(* Logix 5000 project; controller reports 1756-L63 rev 20.11; software revision 20.04; part 11 of 52 *)

        [254].log_data[16].valid := 1, [254].log_data[17].valid := 1, [254].log_data[18].valid := 1, [254].log_data[19].valid := 1, [254].time.Year := 2023, [254].time.Month := 1, [254].time.Day := 18, [254].time.Hour := 21, [254].time.Minute := 34, [254].time.Second := 59, [255].log_data[0].min := 1.0, [255].log_data[0].max := 1.0, [255].log_data[0].total := 300.0, [255].log_data[0].time := 300.0, [255].log_data[0].minminute := 35, [255].log_data[0].maxminute := 35, [255].log_data[0].valid := 1, [255].log_data[1].valid := 1, [255].log_data[2].valid := 1, [255].log_data[3].valid := 1, [255].log_data[4].valid := 1, [255].log_data[5].valid := 1, [255].log_data[6].valid := 1, [255].log_data[7].valid := 1, [255].log_data[8].valid := 1, [255].log_data[9].valid := 1, [255].log_data[10].valid := 1, [255].log_data[11].valid := 1, [255].log_data[12].valid := 1, [255].log_data[13].valid := 1, [255].log_data[14].valid := 1, [255].log_data[15].valid := 1, [255].log_data[16].valid := 1, [255].log_data[17].valid := 1, [255].log_data[18].valid := 1, [255].log_data[19].valid := 1, [255].time.Year := 2023, [255].time.Month := 1, [255].time.Day := 18, [255].time.Hour := 21, [255].time.Minute := 39, [255].time.Second := 59, [256].log_data[0].min := 1.0, [256].log_data[0].max := 1.0, [256].log_data[0].total := 300.0, [256].log_data[0].time := 300.0, [256].log_data[0].minminute := 40, [256].log_data[0].maxminute := 40, [256].log_data[0].valid := 1, [256].log_data[1].valid := 1, [256].log_data[2].valid := 1, [256].log_data[3].valid := 1, [256].log_data[4].valid := 1, [256].log_data[5].valid := 1, [256].log_data[6].valid := 1, [256].log_data[7].valid := 1, [256].log_data[8].valid := 1, [256].log_data[9].valid := 1, [256].log_data[10].valid := 1, [256].log_data[11].valid := 1,
        [256].log_data[12].valid := 1, [256].log_data[13].valid := 1, [256].log_data[14].valid := 1, [256].log_data[15].valid := 1, [256].log_data[16].valid := 1, [256].log_data[17].valid := 1, [256].log_data[18].valid := 1, [256].log_data[19].valid := 1, [256].time.Year := 2023, [256].time.Month := 1, [256].time.Day := 18, [256].time.Hour := 21, [256].time.Minute := 44, [256].time.Second := 59, [257].log_data[0].min := 1.0, [257].log_data[0].max := 1.0, [257].log_data[0].total := 300.0, [257].log_data[0].time := 300.0, [257].log_data[0].minminute := 45, [257].log_data[0].maxminute := 45, [257].log_data[0].valid := 1, [257].log_data[1].valid := 1, [257].log_data[2].valid := 1, [257].log_data[3].valid := 1, [257].log_data[4].valid := 1, [257].log_data[5].valid := 1, [257].log_data[6].valid := 1, [257].log_data[7].valid := 1, [257].log_data[8].valid := 1, [257].log_data[9].valid := 1, [257].log_data[10].valid := 1, [257].log_data[11].valid := 1, [257].log_data[12].valid := 1, [257].log_data[13].valid := 1, [257].log_data[14].valid := 1, [257].log_data[15].valid := 1, [257].log_data[16].valid := 1, [257].log_data[17].valid := 1, [257].log_data[18].valid := 1, [257].log_data[19].valid := 1, [257].time.Year := 2023, [257].time.Month := 1, [257].time.Day := 18, [257].time.Hour := 21, [257].time.Minute := 49, [257].time.Second := 59, [258].log_data[0].min := 1.0, [258].log_data[0].max := 1.0, [258].log_data[0].total := 300.0, [258].log_data[0].time := 300.0, [258].log_data[0].minminute := 50, [258].log_data[0].maxminute := 50, [258].log_data[0].valid := 1, [258].log_data[1].valid := 1, [258].log_data[2].valid := 1, [258].log_data[3].valid := 1, [258].log_data[4].valid := 1, [258].log_data[5].valid := 1, [258].log_data[6].valid := 1, [258].log_data[7].valid := 1,
        [258].log_data[8].valid := 1, [258].log_data[9].valid := 1, [258].log_data[10].valid := 1, [258].log_data[11].valid := 1, [258].log_data[12].valid := 1, [258].log_data[13].valid := 1, [258].log_data[14].valid := 1, [258].log_data[15].valid := 1, [258].log_data[16].valid := 1, [258].log_data[17].valid := 1, [258].log_data[18].valid := 1, [258].log_data[19].valid := 1, [258].time.Year := 2023, [258].time.Month := 1, [258].time.Day := 18, [258].time.Hour := 21, [258].time.Minute := 54, [258].time.Second := 59, [259].log_data[0].min := 1.0, [259].log_data[0].max := 1.0, [259].log_data[0].total := 300.0, [259].log_data[0].time := 300.0, [259].log_data[0].minminute := 55, [259].log_data[0].maxminute := 55, [259].log_data[0].valid := 1, [259].log_data[1].valid := 1, [259].log_data[2].valid := 1, [259].log_data[3].valid := 1, [259].log_data[4].valid := 1, [259].log_data[5].valid := 1, [259].log_data[6].valid := 1, [259].log_data[7].valid := 1, [259].log_data[8].valid := 1, [259].log_data[9].valid := 1, [259].log_data[10].valid := 1, [259].log_data[11].valid := 1, [259].log_data[12].valid := 1, [259].log_data[13].valid := 1, [259].log_data[14].valid := 1, [259].log_data[15].valid := 1, [259].log_data[16].valid := 1, [259].log_data[17].valid := 1, [259].log_data[18].valid := 1, [259].log_data[19].valid := 1, [259].time.Year := 2023, [259].time.Month := 1, [259].time.Day := 18, [259].time.Hour := 21, [259].time.Minute := 59, [259].time.Second := 59, [260].log_data[0].min := 1.0, [260].log_data[0].max := 1.0, [260].log_data[0].total := 300.0, [260].log_data[0].time := 300.0, [260].log_data[0].valid := 1, [260].log_data[1].valid := 1, [260].log_data[2].valid := 1, [260].log_data[3].valid := 1, [260].log_data[4].valid := 1, [260].log_data[5].valid := 1,
        [260].log_data[6].valid := 1, [260].log_data[7].valid := 1, [260].log_data[8].valid := 1, [260].log_data[9].valid := 1, [260].log_data[10].valid := 1, [260].log_data[11].valid := 1, [260].log_data[12].valid := 1, [260].log_data[13].valid := 1, [260].log_data[14].valid := 1, [260].log_data[15].valid := 1, [260].log_data[16].valid := 1, [260].log_data[17].valid := 1, [260].log_data[18].valid := 1, [260].log_data[19].valid := 1, [260].time.Year := 2023, [260].time.Month := 1, [260].time.Day := 18, [260].time.Hour := 22, [260].time.Minute := 4, [260].time.Second := 59, [261].log_data[0].min := 1.0, [261].log_data[0].max := 1.0, [261].log_data[0].total := 300.0, [261].log_data[0].time := 300.0, [261].log_data[0].minminute := 5, [261].log_data[0].maxminute := 5, [261].log_data[0].valid := 1, [261].log_data[1].valid := 1, [261].log_data[2].valid := 1, [261].log_data[3].valid := 1, [261].log_data[4].valid := 1, [261].log_data[5].valid := 1, [261].log_data[6].valid := 1, [261].log_data[7].valid := 1, [261].log_data[8].valid := 1, [261].log_data[9].valid := 1, [261].log_data[10].valid := 1, [261].log_data[11].valid := 1, [261].log_data[12].valid := 1, [261].log_data[13].valid := 1, [261].log_data[14].valid := 1, [261].log_data[15].valid := 1, [261].log_data[16].valid := 1, [261].log_data[17].valid := 1, [261].log_data[18].valid := 1, [261].log_data[19].valid := 1, [261].time.Year := 2023, [261].time.Month := 1, [261].time.Day := 18, [261].time.Hour := 22, [261].time.Minute := 9, [261].time.Second := 59, [262].log_data[0].min := 1.0, [262].log_data[0].max := 1.0, [262].log_data[0].total := 300.0, [262].log_data[0].time := 300.0, [262].log_data[0].minminute := 10, [262].log_data[0].maxminute := 10, [262].log_data[0].valid := 1, [262].log_data[1].valid := 1,
        [262].log_data[2].valid := 1, [262].log_data[3].valid := 1, [262].log_data[4].valid := 1, [262].log_data[5].valid := 1, [262].log_data[6].valid := 1, [262].log_data[7].valid := 1, [262].log_data[8].valid := 1, [262].log_data[9].valid := 1, [262].log_data[10].valid := 1, [262].log_data[11].valid := 1, [262].log_data[12].valid := 1, [262].log_data[13].valid := 1, [262].log_data[14].valid := 1, [262].log_data[15].valid := 1, [262].log_data[16].valid := 1, [262].log_data[17].valid := 1, [262].log_data[18].valid := 1, [262].log_data[19].valid := 1, [262].time.Year := 2023, [262].time.Month := 1, [262].time.Day := 18, [262].time.Hour := 22, [262].time.Minute := 14, [262].time.Second := 59, [263].log_data[0].min := 1.0, [263].log_data[0].max := 1.0, [263].log_data[0].total := 300.0, [263].log_data[0].time := 300.0, [263].log_data[0].minminute := 15, [263].log_data[0].maxminute := 15, [263].log_data[0].valid := 1, [263].log_data[1].valid := 1, [263].log_data[2].valid := 1, [263].log_data[3].valid := 1, [263].log_data[4].valid := 1, [263].log_data[5].valid := 1, [263].log_data[6].valid := 1, [263].log_data[7].valid := 1, [263].log_data[8].valid := 1, [263].log_data[9].valid := 1, [263].log_data[10].valid := 1, [263].log_data[11].valid := 1, [263].log_data[12].valid := 1, [263].log_data[13].valid := 1, [263].log_data[14].valid := 1, [263].log_data[15].valid := 1, [263].log_data[16].valid := 1, [263].log_data[17].valid := 1, [263].log_data[18].valid := 1, [263].log_data[19].valid := 1, [263].time.Year := 2023, [263].time.Month := 1, [263].time.Day := 18, [263].time.Hour := 22, [263].time.Minute := 19, [263].time.Second := 59, [264].log_data[0].min := 1.0, [264].log_data[0].max := 1.0, [264].log_data[0].total := 300.0, [264].log_data[0].time := 300.0,
        [264].log_data[0].minminute := 20, [264].log_data[0].maxminute := 20, [264].log_data[0].valid := 1, [264].log_data[1].valid := 1, [264].log_data[2].valid := 1, [264].log_data[3].valid := 1, [264].log_data[4].valid := 1, [264].log_data[5].valid := 1, [264].log_data[6].valid := 1, [264].log_data[7].valid := 1, [264].log_data[8].valid := 1, [264].log_data[9].valid := 1, [264].log_data[10].valid := 1, [264].log_data[11].valid := 1, [264].log_data[12].valid := 1, [264].log_data[13].valid := 1, [264].log_data[14].valid := 1, [264].log_data[15].valid := 1, [264].log_data[16].valid := 1, [264].log_data[17].valid := 1, [264].log_data[18].valid := 1, [264].log_data[19].valid := 1, [264].time.Year := 2023, [264].time.Month := 1, [264].time.Day := 18, [264].time.Hour := 22, [264].time.Minute := 24, [264].time.Second := 59, [265].log_data[0].min := 1.0, [265].log_data[0].max := 1.0, [265].log_data[0].total := 300.0, [265].log_data[0].time := 300.0, [265].log_data[0].minminute := 25, [265].log_data[0].maxminute := 25, [265].log_data[0].valid := 1, [265].log_data[1].valid := 1, [265].log_data[2].valid := 1, [265].log_data[3].valid := 1, [265].log_data[4].valid := 1, [265].log_data[5].valid := 1, [265].log_data[6].valid := 1, [265].log_data[7].valid := 1, [265].log_data[8].valid := 1, [265].log_data[9].valid := 1, [265].log_data[10].valid := 1, [265].log_data[11].valid := 1, [265].log_data[12].valid := 1, [265].log_data[13].valid := 1, [265].log_data[14].valid := 1, [265].log_data[15].valid := 1, [265].log_data[16].valid := 1, [265].log_data[17].valid := 1, [265].log_data[18].valid := 1, [265].log_data[19].valid := 1, [265].time.Year := 2023, [265].time.Month := 1, [265].time.Day := 18, [265].time.Hour := 22, [265].time.Minute := 29, [265].time.Second := 59,
        [266].log_data[0].min := 1.0, [266].log_data[0].max := 1.0, [266].log_data[0].total := 300.0, [266].log_data[0].time := 300.0, [266].log_data[0].minminute := 30, [266].log_data[0].maxminute := 30, [266].log_data[0].valid := 1, [266].log_data[1].valid := 1, [266].log_data[2].valid := 1, [266].log_data[3].valid := 1, [266].log_data[4].valid := 1, [266].log_data[5].valid := 1, [266].log_data[6].valid := 1, [266].log_data[7].valid := 1, [266].log_data[8].valid := 1, [266].log_data[9].valid := 1, [266].log_data[10].valid := 1, [266].log_data[11].valid := 1, [266].log_data[12].valid := 1, [266].log_data[13].valid := 1, [266].log_data[14].valid := 1, [266].log_data[15].valid := 1, [266].log_data[16].valid := 1, [266].log_data[17].valid := 1, [266].log_data[18].valid := 1, [266].log_data[19].valid := 1, [266].time.Year := 2023, [266].time.Month := 1, [266].time.Day := 18, [266].time.Hour := 22, [266].time.Minute := 34, [266].time.Second := 59, [267].log_data[0].min := 1.0, [267].log_data[0].max := 1.0, [267].log_data[0].total := 300.0, [267].log_data[0].time := 300.0, [267].log_data[0].minminute := 35, [267].log_data[0].maxminute := 35, [267].log_data[0].valid := 1, [267].log_data[1].valid := 1, [267].log_data[2].valid := 1, [267].log_data[3].valid := 1, [267].log_data[4].valid := 1, [267].log_data[5].valid := 1, [267].log_data[6].valid := 1, [267].log_data[7].valid := 1, [267].log_data[8].valid := 1, [267].log_data[9].valid := 1, [267].log_data[10].valid := 1, [267].log_data[11].valid := 1, [267].log_data[12].valid := 1, [267].log_data[13].valid := 1, [267].log_data[14].valid := 1, [267].log_data[15].valid := 1, [267].log_data[16].valid := 1, [267].log_data[17].valid := 1, [267].log_data[18].valid := 1, [267].log_data[19].valid := 1, [267].time.Year := 2023, [267].time.Month := 1,
        [267].time.Day := 18, [267].time.Hour := 22, [267].time.Minute := 39, [267].time.Second := 59, [268].log_data[0].min := 1.0, [268].log_data[0].max := 1.0, [268].log_data[0].total := 300.0, [268].log_data[0].time := 300.0, [268].log_data[0].minminute := 40, [268].log_data[0].maxminute := 40, [268].log_data[0].valid := 1, [268].log_data[1].valid := 1, [268].log_data[2].valid := 1, [268].log_data[3].valid := 1, [268].log_data[4].valid := 1, [268].log_data[5].valid := 1, [268].log_data[6].valid := 1, [268].log_data[7].valid := 1, [268].log_data[8].valid := 1, [268].log_data[9].valid := 1, [268].log_data[10].valid := 1, [268].log_data[11].valid := 1, [268].log_data[12].valid := 1, [268].log_data[13].valid := 1, [268].log_data[14].valid := 1, [268].log_data[15].valid := 1, [268].log_data[16].valid := 1, [268].log_data[17].valid := 1, [268].log_data[18].valid := 1, [268].log_data[19].valid := 1, [268].time.Year := 2023, [268].time.Month := 1, [268].time.Day := 18, [268].time.Hour := 22, [268].time.Minute := 44, [268].time.Second := 59, [269].log_data[0].min := 1.0, [269].log_data[0].max := 1.0, [269].log_data[0].total := 300.0, [269].log_data[0].time := 300.0, [269].log_data[0].minminute := 45, [269].log_data[0].maxminute := 45, [269].log_data[0].valid := 1, [269].log_data[1].valid := 1, [269].log_data[2].valid := 1, [269].log_data[3].valid := 1, [269].log_data[4].valid := 1, [269].log_data[5].valid := 1, [269].log_data[6].valid := 1, [269].log_data[7].valid := 1, [269].log_data[8].valid := 1, [269].log_data[9].valid := 1, [269].log_data[10].valid := 1, [269].log_data[11].valid := 1, [269].log_data[12].valid := 1, [269].log_data[13].valid := 1, [269].log_data[14].valid := 1, [269].log_data[15].valid := 1, [269].log_data[16].valid := 1, [269].log_data[17].valid := 1,
        [269].log_data[18].valid := 1, [269].log_data[19].valid := 1, [269].time.Year := 2023, [269].time.Month := 1, [269].time.Day := 18, [269].time.Hour := 22, [269].time.Minute := 49, [269].time.Second := 59, [270].log_data[0].min := 1.0, [270].log_data[0].max := 1.0, [270].log_data[0].total := 300.0, [270].log_data[0].time := 300.0, [270].log_data[0].minminute := 50, [270].log_data[0].maxminute := 50, [270].log_data[0].valid := 1, [270].log_data[1].valid := 1, [270].log_data[2].valid := 1, [270].log_data[3].valid := 1, [270].log_data[4].valid := 1, [270].log_data[5].valid := 1, [270].log_data[6].valid := 1, [270].log_data[7].valid := 1, [270].log_data[8].valid := 1, [270].log_data[9].valid := 1, [270].log_data[10].valid := 1, [270].log_data[11].valid := 1, [270].log_data[12].valid := 1, [270].log_data[13].valid := 1, [270].log_data[14].valid := 1, [270].log_data[15].valid := 1, [270].log_data[16].valid := 1, [270].log_data[17].valid := 1, [270].log_data[18].valid := 1, [270].log_data[19].valid := 1, [270].time.Year := 2023, [270].time.Month := 1, [270].time.Day := 18, [270].time.Hour := 22, [270].time.Minute := 54, [270].time.Second := 59, [271].log_data[0].min := 1.0, [271].log_data[0].max := 1.0, [271].log_data[0].total := 300.0, [271].log_data[0].time := 300.0, [271].log_data[0].minminute := 55, [271].log_data[0].maxminute := 55, [271].log_data[0].valid := 1, [271].log_data[1].valid := 1, [271].log_data[2].valid := 1, [271].log_data[3].valid := 1, [271].log_data[4].valid := 1, [271].log_data[5].valid := 1, [271].log_data[6].valid := 1, [271].log_data[7].valid := 1, [271].log_data[8].valid := 1, [271].log_data[9].valid := 1, [271].log_data[10].valid := 1, [271].log_data[11].valid := 1, [271].log_data[12].valid := 1, [271].log_data[13].valid := 1,
        [271].log_data[14].valid := 1, [271].log_data[15].valid := 1, [271].log_data[16].valid := 1, [271].log_data[17].valid := 1, [271].log_data[18].valid := 1, [271].log_data[19].valid := 1, [271].time.Year := 2023, [271].time.Month := 1, [271].time.Day := 18, [271].time.Hour := 22, [271].time.Minute := 59, [271].time.Second := 59, [272].log_data[0].min := 1.0, [272].log_data[0].max := 1.0, [272].log_data[0].total := 300.0, [272].log_data[0].time := 300.0, [272].log_data[0].valid := 1, [272].log_data[1].valid := 1, [272].log_data[2].valid := 1, [272].log_data[3].valid := 1, [272].log_data[4].valid := 1, [272].log_data[5].valid := 1, [272].log_data[6].valid := 1, [272].log_data[7].valid := 1, [272].log_data[8].valid := 1, [272].log_data[9].valid := 1, [272].log_data[10].valid := 1, [272].log_data[11].valid := 1, [272].log_data[12].valid := 1, [272].log_data[13].valid := 1, [272].log_data[14].valid := 1, [272].log_data[15].valid := 1, [272].log_data[16].valid := 1, [272].log_data[17].valid := 1, [272].log_data[18].valid := 1, [272].log_data[19].valid := 1, [272].time.Year := 2023, [272].time.Month := 1, [272].time.Day := 18, [272].time.Hour := 23, [272].time.Minute := 4, [272].time.Second := 59, [273].log_data[0].min := 1.0, [273].log_data[0].max := 1.0, [273].log_data[0].total := 300.0, [273].log_data[0].time := 300.0, [273].log_data[0].minminute := 5, [273].log_data[0].maxminute := 5, [273].log_data[0].valid := 1, [273].log_data[1].valid := 1, [273].log_data[2].valid := 1, [273].log_data[3].valid := 1, [273].log_data[4].valid := 1, [273].log_data[5].valid := 1, [273].log_data[6].valid := 1, [273].log_data[7].valid := 1, [273].log_data[8].valid := 1, [273].log_data[9].valid := 1, [273].log_data[10].valid := 1, [273].log_data[11].valid := 1,
        [273].log_data[12].valid := 1, [273].log_data[13].valid := 1, [273].log_data[14].valid := 1, [273].log_data[15].valid := 1, [273].log_data[16].valid := 1, [273].log_data[17].valid := 1, [273].log_data[18].valid := 1, [273].log_data[19].valid := 1, [273].time.Year := 2023, [273].time.Month := 1, [273].time.Day := 18, [273].time.Hour := 23, [273].time.Minute := 9, [273].time.Second := 59, [274].log_data[0].min := 1.0, [274].log_data[0].max := 1.0, [274].log_data[0].total := 300.0, [274].log_data[0].time := 300.0, [274].log_data[0].minminute := 10, [274].log_data[0].maxminute := 10, [274].log_data[0].valid := 1, [274].log_data[1].valid := 1, [274].log_data[2].valid := 1, [274].log_data[3].valid := 1, [274].log_data[4].valid := 1, [274].log_data[5].valid := 1, [274].log_data[6].valid := 1, [274].log_data[7].valid := 1, [274].log_data[8].valid := 1, [274].log_data[9].valid := 1, [274].log_data[10].valid := 1, [274].log_data[11].valid := 1, [274].log_data[12].valid := 1, [274].log_data[13].valid := 1, [274].log_data[14].valid := 1, [274].log_data[15].valid := 1, [274].log_data[16].valid := 1, [274].log_data[17].valid := 1, [274].log_data[18].valid := 1, [274].log_data[19].valid := 1, [274].time.Year := 2023, [274].time.Month := 1, [274].time.Day := 18, [274].time.Hour := 23, [274].time.Minute := 14, [274].time.Second := 59, [275].log_data[0].min := 1.0, [275].log_data[0].max := 1.0, [275].log_data[0].total := 300.0, [275].log_data[0].time := 300.0, [275].log_data[0].minminute := 15, [275].log_data[0].maxminute := 15, [275].log_data[0].valid := 1, [275].log_data[1].valid := 1, [275].log_data[2].valid := 1, [275].log_data[3].valid := 1, [275].log_data[4].valid := 1, [275].log_data[5].valid := 1, [275].log_data[6].valid := 1, [275].log_data[7].valid := 1,
        [275].log_data[8].valid := 1, [275].log_data[9].valid := 1, [275].log_data[10].valid := 1, [275].log_data[11].valid := 1, [275].log_data[12].valid := 1, [275].log_data[13].valid := 1, [275].log_data[14].valid := 1, [275].log_data[15].valid := 1, [275].log_data[16].valid := 1, [275].log_data[17].valid := 1, [275].log_data[18].valid := 1, [275].log_data[19].valid := 1, [275].time.Year := 2023, [275].time.Month := 1, [275].time.Day := 18, [275].time.Hour := 23, [275].time.Minute := 19, [275].time.Second := 59, [276].log_data[0].min := 1.0, [276].log_data[0].max := 1.0, [276].log_data[0].total := 300.0, [276].log_data[0].time := 300.0, [276].log_data[0].minminute := 20, [276].log_data[0].maxminute := 20, [276].log_data[0].valid := 1, [276].log_data[1].valid := 1, [276].log_data[2].valid := 1, [276].log_data[3].valid := 1, [276].log_data[4].valid := 1, [276].log_data[5].valid := 1, [276].log_data[6].valid := 1, [276].log_data[7].valid := 1, [276].log_data[8].valid := 1, [276].log_data[9].valid := 1, [276].log_data[10].valid := 1, [276].log_data[11].valid := 1, [276].log_data[12].valid := 1, [276].log_data[13].valid := 1, [276].log_data[14].valid := 1, [276].log_data[15].valid := 1, [276].log_data[16].valid := 1, [276].log_data[17].valid := 1, [276].log_data[18].valid := 1, [276].log_data[19].valid := 1, [276].time.Year := 2023, [276].time.Month := 1, [276].time.Day := 18, [276].time.Hour := 23, [276].time.Minute := 24, [276].time.Second := 59, [277].log_data[0].min := 1.0, [277].log_data[0].max := 1.0, [277].log_data[0].total := 300.0, [277].log_data[0].time := 300.0, [277].log_data[0].minminute := 25, [277].log_data[0].maxminute := 25, [277].log_data[0].valid := 1, [277].log_data[1].valid := 1, [277].log_data[2].valid := 1, [277].log_data[3].valid := 1,
        [277].log_data[4].valid := 1, [277].log_data[5].valid := 1, [277].log_data[6].valid := 1, [277].log_data[7].valid := 1, [277].log_data[8].valid := 1, [277].log_data[9].valid := 1, [277].log_data[10].valid := 1, [277].log_data[11].valid := 1, [277].log_data[12].valid := 1, [277].log_data[13].valid := 1, [277].log_data[14].valid := 1, [277].log_data[15].valid := 1, [277].log_data[16].valid := 1, [277].log_data[17].valid := 1, [277].log_data[18].valid := 1, [277].log_data[19].valid := 1, [277].time.Year := 2023, [277].time.Month := 1, [277].time.Day := 18, [277].time.Hour := 23, [277].time.Minute := 29, [277].time.Second := 59, [278].log_data[0].min := 1.0, [278].log_data[0].max := 1.0, [278].log_data[0].total := 300.0, [278].log_data[0].time := 300.0, [278].log_data[0].minminute := 30, [278].log_data[0].maxminute := 30, [278].log_data[0].valid := 1, [278].log_data[1].valid := 1, [278].log_data[2].valid := 1, [278].log_data[3].valid := 1, [278].log_data[4].valid := 1, [278].log_data[5].valid := 1, [278].log_data[6].valid := 1, [278].log_data[7].valid := 1, [278].log_data[8].valid := 1, [278].log_data[9].valid := 1, [278].log_data[10].valid := 1, [278].log_data[11].valid := 1, [278].log_data[12].valid := 1, [278].log_data[13].valid := 1, [278].log_data[14].valid := 1, [278].log_data[15].valid := 1, [278].log_data[16].valid := 1, [278].log_data[17].valid := 1, [278].log_data[18].valid := 1, [278].log_data[19].valid := 1, [278].time.Year := 2023, [278].time.Month := 1, [278].time.Day := 18, [278].time.Hour := 23, [278].time.Minute := 34, [278].time.Second := 59, [279].log_data[0].min := 1.0, [279].log_data[0].max := 1.0, [279].log_data[0].total := 300.0, [279].log_data[0].time := 300.0, [279].log_data[0].minminute := 35, [279].log_data[0].maxminute := 35,
        [279].log_data[0].valid := 1, [279].log_data[1].valid := 1, [279].log_data[2].valid := 1, [279].log_data[3].valid := 1, [279].log_data[4].valid := 1, [279].log_data[5].valid := 1, [279].log_data[6].valid := 1, [279].log_data[7].valid := 1, [279].log_data[8].valid := 1, [279].log_data[9].valid := 1, [279].log_data[10].valid := 1, [279].log_data[11].valid := 1, [279].log_data[12].valid := 1, [279].log_data[13].valid := 1, [279].log_data[14].valid := 1, [279].log_data[15].valid := 1, [279].log_data[16].valid := 1, [279].log_data[17].valid := 1, [279].log_data[18].valid := 1, [279].log_data[19].valid := 1, [279].time.Year := 2023, [279].time.Month := 1, [279].time.Day := 18, [279].time.Hour := 23, [279].time.Minute := 39, [279].time.Second := 59, [280].log_data[0].min := 1.0, [280].log_data[0].max := 1.0, [280].log_data[0].total := 300.0, [280].log_data[0].time := 300.0, [280].log_data[0].minminute := 40, [280].log_data[0].maxminute := 40, [280].log_data[0].valid := 1, [280].log_data[1].valid := 1, [280].log_data[2].valid := 1, [280].log_data[3].valid := 1, [280].log_data[4].valid := 1, [280].log_data[5].valid := 1, [280].log_data[6].valid := 1, [280].log_data[7].valid := 1, [280].log_data[8].valid := 1, [280].log_data[9].valid := 1, [280].log_data[10].valid := 1, [280].log_data[11].valid := 1, [280].log_data[12].valid := 1, [280].log_data[13].valid := 1, [280].log_data[14].valid := 1, [280].log_data[15].valid := 1, [280].log_data[16].valid := 1, [280].log_data[17].valid := 1, [280].log_data[18].valid := 1, [280].log_data[19].valid := 1, [280].time.Year := 2023, [280].time.Month := 1, [280].time.Day := 18, [280].time.Hour := 23, [280].time.Minute := 44, [280].time.Second := 59, [281].log_data[0].min := 1.0, [281].log_data[0].max := 1.0,
        [281].log_data[0].total := 300.0, [281].log_data[0].time := 300.0, [281].log_data[0].minminute := 45, [281].log_data[0].maxminute := 45, [281].log_data[0].valid := 1, [281].log_data[1].valid := 1, [281].log_data[2].valid := 1, [281].log_data[3].valid := 1, [281].log_data[4].valid := 1, [281].log_data[5].valid := 1, [281].log_data[6].valid := 1, [281].log_data[7].valid := 1, [281].log_data[8].valid := 1, [281].log_data[9].valid := 1, [281].log_data[10].valid := 1, [281].log_data[11].valid := 1, [281].log_data[12].valid := 1, [281].log_data[13].valid := 1, [281].log_data[14].valid := 1, [281].log_data[15].valid := 1, [281].log_data[16].valid := 1, [281].log_data[17].valid := 1, [281].log_data[18].valid := 1, [281].log_data[19].valid := 1, [281].time.Year := 2023, [281].time.Month := 1, [281].time.Day := 18, [281].time.Hour := 23, [281].time.Minute := 49, [281].time.Second := 59, [282].log_data[0].min := 1.0, [282].log_data[0].max := 1.0, [282].log_data[0].total := 300.0, [282].log_data[0].time := 300.0, [282].log_data[0].minminute := 50, [282].log_data[0].maxminute := 50, [282].log_data[0].valid := 1, [282].log_data[1].valid := 1, [282].log_data[2].valid := 1, [282].log_data[3].valid := 1, [282].log_data[4].valid := 1, [282].log_data[5].valid := 1, [282].log_data[6].valid := 1, [282].log_data[7].valid := 1, [282].log_data[8].valid := 1, [282].log_data[9].valid := 1, [282].log_data[10].valid := 1, [282].log_data[11].valid := 1, [282].log_data[12].valid := 1, [282].log_data[13].valid := 1, [282].log_data[14].valid := 1, [282].log_data[15].valid := 1, [282].log_data[16].valid := 1, [282].log_data[17].valid := 1, [282].log_data[18].valid := 1, [282].log_data[19].valid := 1, [282].time.Year := 2023, [282].time.Month := 1, [282].time.Day := 18, [282].time.Hour := 23,
        [282].time.Minute := 54, [282].time.Second := 59, [283].log_data[0].min := 1.0, [283].log_data[0].max := 1.0, [283].log_data[0].total := 300.0, [283].log_data[0].time := 300.0, [283].log_data[0].minminute := 55, [283].log_data[0].maxminute := 55, [283].log_data[0].valid := 1, [283].log_data[1].valid := 1, [283].log_data[2].valid := 1, [283].log_data[3].valid := 1, [283].log_data[4].valid := 1, [283].log_data[5].valid := 1, [283].log_data[6].valid := 1, [283].log_data[7].valid := 1, [283].log_data[8].valid := 1, [283].log_data[9].valid := 1, [283].log_data[10].valid := 1, [283].log_data[11].valid := 1, [283].log_data[12].valid := 1, [283].log_data[13].valid := 1, [283].log_data[14].valid := 1, [283].log_data[15].valid := 1, [283].log_data[16].valid := 1, [283].log_data[17].valid := 1, [283].log_data[18].valid := 1, [283].log_data[19].valid := 1, [283].time.Year := 2023, [283].time.Month := 1, [283].time.Day := 18, [283].time.Hour := 23, [283].time.Minute := 59, [283].time.Second := 59, [284].log_data[0].min := 1.0, [284].log_data[0].max := 1.0, [284].log_data[0].total := 300.0, [284].log_data[0].time := 300.0, [284].log_data[0].valid := 1, [284].log_data[1].valid := 1, [284].log_data[2].valid := 1, [284].log_data[3].valid := 1, [284].log_data[4].valid := 1, [284].log_data[5].valid := 1, [284].log_data[6].valid := 1, [284].log_data[7].valid := 1, [284].log_data[8].valid := 1, [284].log_data[9].valid := 1, [284].log_data[10].valid := 1, [284].log_data[11].valid := 1, [284].log_data[12].valid := 1, [284].log_data[13].valid := 1, [284].log_data[14].valid := 1, [284].log_data[15].valid := 1, [284].log_data[16].valid := 1, [284].log_data[17].valid := 1, [284].log_data[18].valid := 1, [284].log_data[19].valid := 1, [284].time.Year := 2023, [284].time.Month := 1,
        [284].time.Day := 19, [284].time.Minute := 4, [284].time.Second := 59, [285].log_data[0].min := 1.0, [285].log_data[0].max := 1.0, [285].log_data[0].total := 300.0, [285].log_data[0].time := 300.0, [285].log_data[0].minminute := 5, [285].log_data[0].maxminute := 5, [285].log_data[0].valid := 1, [285].log_data[1].valid := 1, [285].log_data[2].valid := 1, [285].log_data[3].valid := 1, [285].log_data[4].valid := 1, [285].log_data[5].valid := 1, [285].log_data[6].valid := 1, [285].log_data[7].valid := 1, [285].log_data[8].valid := 1, [285].log_data[9].valid := 1, [285].log_data[10].valid := 1, [285].log_data[11].valid := 1, [285].log_data[12].valid := 1, [285].log_data[13].valid := 1, [285].log_data[14].valid := 1, [285].log_data[15].valid := 1, [285].log_data[16].valid := 1, [285].log_data[17].valid := 1, [285].log_data[18].valid := 1, [285].log_data[19].valid := 1, [285].time.Year := 2023, [285].time.Month := 1, [285].time.Day := 19, [285].time.Minute := 9, [285].time.Second := 59, [286].log_data[0].min := 1.0, [286].log_data[0].max := 1.0, [286].log_data[0].total := 300.0, [286].log_data[0].time := 300.0, [286].log_data[0].minminute := 10, [286].log_data[0].maxminute := 10, [286].log_data[0].valid := 1, [286].log_data[1].valid := 1, [286].log_data[2].valid := 1, [286].log_data[3].valid := 1, [286].log_data[4].valid := 1, [286].log_data[5].valid := 1, [286].log_data[6].valid := 1, [286].log_data[7].valid := 1, [286].log_data[8].valid := 1, [286].log_data[9].valid := 1, [286].log_data[10].valid := 1, [286].log_data[11].valid := 1, [286].log_data[12].valid := 1, [286].log_data[13].valid := 1, [286].log_data[14].valid := 1, [286].log_data[15].valid := 1, [286].log_data[16].valid := 1, [286].log_data[17].valid := 1, [286].log_data[18].valid := 1, [286].log_data[19].valid := 1,
        [286].time.Year := 2023, [286].time.Month := 1, [286].time.Day := 19, [286].time.Minute := 14, [286].time.Second := 59, [287].log_data[0].min := 1.0, [287].log_data[0].max := 1.0, [287].log_data[0].total := 300.0, [287].log_data[0].time := 300.0, [287].log_data[0].minminute := 15, [287].log_data[0].maxminute := 15, [287].log_data[0].valid := 1, [287].log_data[1].valid := 1, [287].log_data[2].valid := 1, [287].log_data[3].valid := 1, [287].log_data[4].valid := 1, [287].log_data[5].valid := 1, [287].log_data[6].valid := 1, [287].log_data[7].valid := 1, [287].log_data[8].valid := 1, [287].log_data[9].valid := 1, [287].log_data[10].valid := 1, [287].log_data[11].valid := 1, [287].log_data[12].valid := 1, [287].log_data[13].valid := 1, [287].log_data[14].valid := 1, [287].log_data[15].valid := 1, [287].log_data[16].valid := 1, [287].log_data[17].valid := 1, [287].log_data[18].valid := 1, [287].log_data[19].valid := 1, [287].time.Year := 2023, [287].time.Month := 1, [287].time.Day := 19, [287].time.Minute := 19, [287].time.Second := 59, [288].log_data[0].min := 1.0, [288].log_data[0].max := 1.0, [288].log_data[0].total := 300.0, [288].log_data[0].time := 300.0, [288].log_data[0].minminute := 20, [288].log_data[0].maxminute := 20, [288].log_data[0].valid := 1, [288].log_data[1].valid := 1, [288].log_data[2].valid := 1, [288].log_data[3].valid := 1, [288].log_data[4].valid := 1, [288].log_data[5].valid := 1, [288].log_data[6].valid := 1, [288].log_data[7].valid := 1, [288].log_data[8].valid := 1, [288].log_data[9].valid := 1, [288].log_data[10].valid := 1, [288].log_data[11].valid := 1, [288].log_data[12].valid := 1, [288].log_data[13].valid := 1, [288].log_data[14].valid := 1, [288].log_data[15].valid := 1, [288].log_data[16].valid := 1, [288].log_data[17].valid := 1,
        [288].log_data[18].valid := 1, [288].log_data[19].valid := 1, [288].time.Year := 2023, [288].time.Month := 1, [288].time.Day := 19, [288].time.Minute := 24, [288].time.Second := 59, [289].log_data[0].min := 1.0, [289].log_data[0].max := 1.0, [289].log_data[0].total := 300.0, [289].log_data[0].time := 300.0, [289].log_data[0].minminute := 25, [289].log_data[0].maxminute := 25, [289].log_data[0].valid := 1, [289].log_data[1].valid := 1, [289].log_data[2].valid := 1, [289].log_data[3].valid := 1, [289].log_data[4].valid := 1, [289].log_data[5].valid := 1, [289].log_data[6].valid := 1, [289].log_data[7].valid := 1, [289].log_data[8].valid := 1, [289].log_data[9].valid := 1, [289].log_data[10].valid := 1, [289].log_data[11].valid := 1, [289].log_data[12].valid := 1, [289].log_data[13].valid := 1, [289].log_data[14].valid := 1, [289].log_data[15].valid := 1, [289].log_data[16].valid := 1, [289].log_data[17].valid := 1, [289].log_data[18].valid := 1, [289].log_data[19].valid := 1, [289].time.Year := 2023, [289].time.Month := 1, [289].time.Day := 19, [289].time.Minute := 29, [289].time.Second := 59, [290].log_data[0].min := 1.0, [290].log_data[0].max := 1.0, [290].log_data[0].total := 300.0, [290].log_data[0].time := 300.0, [290].log_data[0].minminute := 30, [290].log_data[0].maxminute := 30, [290].log_data[0].valid := 1, [290].log_data[1].valid := 1, [290].log_data[2].valid := 1, [290].log_data[3].valid := 1, [290].log_data[4].valid := 1, [290].log_data[5].valid := 1, [290].log_data[6].valid := 1, [290].log_data[7].valid := 1, [290].log_data[8].valid := 1, [290].log_data[9].valid := 1, [290].log_data[10].valid := 1, [290].log_data[11].valid := 1, [290].log_data[12].valid := 1, [290].log_data[13].valid := 1, [290].log_data[14].valid := 1, [290].log_data[15].valid := 1,
        [290].log_data[16].valid := 1, [290].log_data[17].valid := 1, [290].log_data[18].valid := 1, [290].log_data[19].valid := 1, [290].time.Year := 2023, [290].time.Month := 1, [290].time.Day := 19, [290].time.Minute := 34, [290].time.Second := 59, [291].log_data[0].min := 1.0, [291].log_data[0].max := 1.0, [291].log_data[0].total := 300.0, [291].log_data[0].time := 300.0, [291].log_data[0].minminute := 35, [291].log_data[0].maxminute := 35, [291].log_data[0].valid := 1, [291].log_data[1].valid := 1, [291].log_data[2].valid := 1, [291].log_data[3].valid := 1, [291].log_data[4].valid := 1, [291].log_data[5].valid := 1, [291].log_data[6].valid := 1, [291].log_data[7].valid := 1, [291].log_data[8].valid := 1, [291].log_data[9].valid := 1, [291].log_data[10].valid := 1, [291].log_data[11].valid := 1, [291].log_data[12].valid := 1, [291].log_data[13].valid := 1, [291].log_data[14].valid := 1, [291].log_data[15].valid := 1, [291].log_data[16].valid := 1, [291].log_data[17].valid := 1, [291].log_data[18].valid := 1, [291].log_data[19].valid := 1, [291].time.Year := 2023, [291].time.Month := 1, [291].time.Day := 19, [291].time.Minute := 39, [291].time.Second := 59, [292].log_data[0].min := 1.0, [292].log_data[0].max := 1.0, [292].log_data[0].total := 300.0, [292].log_data[0].time := 300.0, [292].log_data[0].minminute := 40, [292].log_data[0].maxminute := 40, [292].log_data[0].valid := 1, [292].log_data[1].valid := 1, [292].log_data[2].valid := 1, [292].log_data[3].valid := 1, [292].log_data[4].valid := 1, [292].log_data[5].valid := 1, [292].log_data[6].valid := 1, [292].log_data[7].valid := 1, [292].log_data[8].valid := 1, [292].log_data[9].valid := 1, [292].log_data[10].valid := 1, [292].log_data[11].valid := 1, [292].log_data[12].valid := 1, [292].log_data[13].valid := 1,
        [292].log_data[14].valid := 1, [292].log_data[15].valid := 1, [292].log_data[16].valid := 1, [292].log_data[17].valid := 1, [292].log_data[18].valid := 1, [292].log_data[19].valid := 1, [292].time.Year := 2023, [292].time.Month := 1, [292].time.Day := 19, [292].time.Minute := 44, [292].time.Second := 59, [293].log_data[0].min := 1.0, [293].log_data[0].max := 1.0, [293].log_data[0].total := 300.0, [293].log_data[0].time := 300.0, [293].log_data[0].minminute := 45, [293].log_data[0].maxminute := 45, [293].log_data[0].valid := 1, [293].log_data[1].valid := 1, [293].log_data[2].valid := 1, [293].log_data[3].valid := 1, [293].log_data[4].valid := 1, [293].log_data[5].valid := 1, [293].log_data[6].valid := 1, [293].log_data[7].valid := 1, [293].log_data[8].valid := 1, [293].log_data[9].valid := 1, [293].log_data[10].valid := 1, [293].log_data[11].valid := 1, [293].log_data[12].valid := 1, [293].log_data[13].valid := 1, [293].log_data[14].valid := 1, [293].log_data[15].valid := 1, [293].log_data[16].valid := 1, [293].log_data[17].valid := 1, [293].log_data[18].valid := 1, [293].log_data[19].valid := 1, [293].time.Year := 2023, [293].time.Month := 1, [293].time.Day := 19, [293].time.Minute := 49, [293].time.Second := 59, [294].log_data[0].min := 1.0, [294].log_data[0].max := 1.0, [294].log_data[0].total := 300.0, [294].log_data[0].time := 300.0, [294].log_data[0].minminute := 50, [294].log_data[0].maxminute := 50, [294].log_data[0].valid := 1, [294].log_data[1].valid := 1, [294].log_data[2].valid := 1, [294].log_data[3].valid := 1, [294].log_data[4].valid := 1, [294].log_data[5].valid := 1, [294].log_data[6].valid := 1, [294].log_data[7].valid := 1, [294].log_data[8].valid := 1, [294].log_data[9].valid := 1, [294].log_data[10].valid := 1, [294].log_data[11].valid := 1,
        [294].log_data[12].valid := 1, [294].log_data[13].valid := 1, [294].log_data[14].valid := 1, [294].log_data[15].valid := 1, [294].log_data[16].valid := 1, [294].log_data[17].valid := 1, [294].log_data[18].valid := 1, [294].log_data[19].valid := 1, [294].time.Year := 2023, [294].time.Month := 1, [294].time.Day := 19, [294].time.Minute := 54, [294].time.Second := 59, [295].log_data[0].min := 1.0, [295].log_data[0].max := 1.0, [295].log_data[0].total := 300.0, [295].log_data[0].time := 300.0, [295].log_data[0].minminute := 55, [295].log_data[0].maxminute := 55, [295].log_data[0].valid := 1, [295].log_data[1].valid := 1, [295].log_data[2].valid := 1, [295].log_data[3].valid := 1, [295].log_data[4].valid := 1, [295].log_data[5].valid := 1, [295].log_data[6].valid := 1, [295].log_data[7].valid := 1, [295].log_data[8].valid := 1, [295].log_data[9].valid := 1, [295].log_data[10].valid := 1, [295].log_data[11].valid := 1, [295].log_data[12].valid := 1, [295].log_data[13].valid := 1, [295].log_data[14].valid := 1, [295].log_data[15].valid := 1, [295].log_data[16].valid := 1, [295].log_data[17].valid := 1, [295].log_data[18].valid := 1, [295].log_data[19].valid := 1, [295].time.Year := 2023, [295].time.Month := 1, [295].time.Day := 19, [295].time.Minute := 59, [295].time.Second := 59, [296].log_data[0].min := 1.0, [296].log_data[0].max := 1.0, [296].log_data[0].total := 300.0, [296].log_data[0].time := 300.0, [296].log_data[0].valid := 1, [296].log_data[1].valid := 1, [296].log_data[2].valid := 1, [296].log_data[3].valid := 1, [296].log_data[4].valid := 1, [296].log_data[5].valid := 1, [296].log_data[6].valid := 1, [296].log_data[7].valid := 1, [296].log_data[8].valid := 1, [296].log_data[9].valid := 1, [296].log_data[10].valid := 1, [296].log_data[11].valid := 1,
        [296].log_data[12].valid := 1, [296].log_data[13].valid := 1, [296].log_data[14].valid := 1, [296].log_data[15].valid := 1, [296].log_data[16].valid := 1, [296].log_data[17].valid := 1, [296].log_data[18].valid := 1, [296].log_data[19].valid := 1, [296].time.Year := 2023, [296].time.Month := 1, [296].time.Day := 19, [296].time.Hour := 1, [296].time.Minute := 4, [296].time.Second := 59, [297].log_data[0].min := 1.0, [297].log_data[0].max := 1.0, [297].log_data[0].total := 300.0, [297].log_data[0].time := 300.0, [297].log_data[0].minminute := 5, [297].log_data[0].maxminute := 5, [297].log_data[0].valid := 1, [297].log_data[1].valid := 1, [297].log_data[2].valid := 1, [297].log_data[3].valid := 1, [297].log_data[4].valid := 1, [297].log_data[5].valid := 1, [297].log_data[6].valid := 1, [297].log_data[7].valid := 1, [297].log_data[8].valid := 1, [297].log_data[9].valid := 1, [297].log_data[10].valid := 1, [297].log_data[11].valid := 1, [297].log_data[12].valid := 1, [297].log_data[13].valid := 1, [297].log_data[14].valid := 1, [297].log_data[15].valid := 1, [297].log_data[16].valid := 1, [297].log_data[17].valid := 1, [297].log_data[18].valid := 1, [297].log_data[19].valid := 1, [297].time.Year := 2023, [297].time.Month := 1, [297].time.Day := 19, [297].time.Hour := 1, [297].time.Minute := 9, [297].time.Second := 59, [298].log_data[0].min := 1.0, [298].log_data[0].max := 1.0, [298].log_data[0].total := 300.0, [298].log_data[0].time := 300.0, [298].log_data[0].minminute := 10, [298].log_data[0].maxminute := 10, [298].log_data[0].valid := 1, [298].log_data[1].valid := 1, [298].log_data[2].valid := 1, [298].log_data[3].valid := 1, [298].log_data[4].valid := 1, [298].log_data[5].valid := 1, [298].log_data[6].valid := 1, [298].log_data[7].valid := 1,
        [298].log_data[8].valid := 1, [298].log_data[9].valid := 1, [298].log_data[10].valid := 1, [298].log_data[11].valid := 1, [298].log_data[12].valid := 1, [298].log_data[13].valid := 1, [298].log_data[14].valid := 1, [298].log_data[15].valid := 1, [298].log_data[16].valid := 1, [298].log_data[17].valid := 1, [298].log_data[18].valid := 1, [298].log_data[19].valid := 1, [298].time.Year := 2023, [298].time.Month := 1, [298].time.Day := 19, [298].time.Hour := 1, [298].time.Minute := 14, [298].time.Second := 59, [299].log_data[0].min := 1.0, [299].log_data[0].max := 1.0, [299].log_data[0].total := 300.0, [299].log_data[0].time := 300.0, [299].log_data[0].minminute := 15, [299].log_data[0].maxminute := 15, [299].log_data[0].valid := 1, [299].log_data[1].valid := 1, [299].log_data[2].valid := 1, [299].log_data[3].valid := 1, [299].log_data[4].valid := 1, [299].log_data[5].valid := 1, [299].log_data[6].valid := 1, [299].log_data[7].valid := 1, [299].log_data[8].valid := 1, [299].log_data[9].valid := 1, [299].log_data[10].valid := 1, [299].log_data[11].valid := 1, [299].log_data[12].valid := 1, [299].log_data[13].valid := 1, [299].log_data[14].valid := 1, [299].log_data[15].valid := 1, [299].log_data[16].valid := 1, [299].log_data[17].valid := 1, [299].log_data[18].valid := 1, [299].log_data[19].valid := 1, [299].time.Year := 2023, [299].time.Month := 1, [299].time.Day := 19, [299].time.Hour := 1, [299].time.Minute := 19, [299].time.Second := 59, [300].log_data[0].min := 1.0, [300].log_data[0].max := 1.0, [300].log_data[0].total := 300.0, [300].log_data[0].time := 300.0, [300].log_data[0].minminute := 20, [300].log_data[0].maxminute := 20, [300].log_data[0].valid := 1, [300].log_data[1].valid := 1, [300].log_data[2].valid := 1, [300].log_data[3].valid := 1,
        [300].log_data[4].valid := 1, [300].log_data[5].valid := 1, [300].log_data[6].valid := 1, [300].log_data[7].valid := 1, [300].log_data[8].valid := 1, [300].log_data[9].valid := 1, [300].log_data[10].valid := 1, [300].log_data[11].valid := 1, [300].log_data[12].valid := 1, [300].log_data[13].valid := 1, [300].log_data[14].valid := 1, [300].log_data[15].valid := 1, [300].log_data[16].valid := 1, [300].log_data[17].valid := 1, [300].log_data[18].valid := 1, [300].log_data[19].valid := 1, [300].time.Year := 2023, [300].time.Month := 1, [300].time.Day := 19, [300].time.Hour := 1, [300].time.Minute := 24, [300].time.Second := 59, [301].log_data[0].min := 1.0, [301].log_data[0].max := 1.0, [301].log_data[0].total := 300.0, [301].log_data[0].time := 300.0, [301].log_data[0].minminute := 25, [301].log_data[0].maxminute := 25, [301].log_data[0].valid := 1, [301].log_data[1].valid := 1, [301].log_data[2].valid := 1, [301].log_data[3].valid := 1, [301].log_data[4].valid := 1, [301].log_data[5].valid := 1, [301].log_data[6].valid := 1, [301].log_data[7].valid := 1, [301].log_data[8].valid := 1, [301].log_data[9].valid := 1, [301].log_data[10].valid := 1, [301].log_data[11].valid := 1, [301].log_data[12].valid := 1, [301].log_data[13].valid := 1, [301].log_data[14].valid := 1, [301].log_data[15].valid := 1, [301].log_data[16].valid := 1, [301].log_data[17].valid := 1, [301].log_data[18].valid := 1, [301].log_data[19].valid := 1, [301].time.Year := 2023, [301].time.Month := 1, [301].time.Day := 19, [301].time.Hour := 1, [301].time.Minute := 29, [301].time.Second := 59, [302].log_data[0].min := 1.0, [302].log_data[0].max := 1.0, [302].log_data[0].total := 300.0, [302].log_data[0].time := 300.0, [302].log_data[0].minminute := 30, [302].log_data[0].maxminute := 30,
        [302].log_data[0].valid := 1, [302].log_data[1].valid := 1, [302].log_data[2].valid := 1, [302].log_data[3].valid := 1, [302].log_data[4].valid := 1, [302].log_data[5].valid := 1, [302].log_data[6].valid := 1, [302].log_data[7].valid := 1, [302].log_data[8].valid := 1, [302].log_data[9].valid := 1, [302].log_data[10].valid := 1, [302].log_data[11].valid := 1, [302].log_data[12].valid := 1, [302].log_data[13].valid := 1, [302].log_data[14].valid := 1, [302].log_data[15].valid := 1, [302].log_data[16].valid := 1, [302].log_data[17].valid := 1, [302].log_data[18].valid := 1, [302].log_data[19].valid := 1, [302].time.Year := 2023, [302].time.Month := 1, [302].time.Day := 19, [302].time.Hour := 1, [302].time.Minute := 34, [302].time.Second := 59, [303].log_data[0].min := 1.0, [303].log_data[0].max := 1.0, [303].log_data[0].total := 300.0, [303].log_data[0].time := 300.0, [303].log_data[0].minminute := 35, [303].log_data[0].maxminute := 35, [303].log_data[0].valid := 1, [303].log_data[1].valid := 1, [303].log_data[2].valid := 1, [303].log_data[3].valid := 1, [303].log_data[4].valid := 1, [303].log_data[5].valid := 1, [303].log_data[6].valid := 1, [303].log_data[7].valid := 1, [303].log_data[8].valid := 1, [303].log_data[9].valid := 1, [303].log_data[10].valid := 1, [303].log_data[11].valid := 1, [303].log_data[12].valid := 1, [303].log_data[13].valid := 1, [303].log_data[14].valid := 1, [303].log_data[15].valid := 1, [303].log_data[16].valid := 1, [303].log_data[17].valid := 1, [303].log_data[18].valid := 1, [303].log_data[19].valid := 1, [303].time.Year := 2023, [303].time.Month := 1, [303].time.Day := 19, [303].time.Hour := 1, [303].time.Minute := 39, [303].time.Second := 59, [304].log_data[0].min := 1.0, [304].log_data[0].max := 1.0,
        [304].log_data[0].total := 300.0, [304].log_data[0].time := 300.0, [304].log_data[0].minminute := 40, [304].log_data[0].maxminute := 40, [304].log_data[0].valid := 1, [304].log_data[1].valid := 1, [304].log_data[2].valid := 1, [304].log_data[3].valid := 1, [304].log_data[4].valid := 1, [304].log_data[5].valid := 1, [304].log_data[6].valid := 1, [304].log_data[7].valid := 1, [304].log_data[8].valid := 1, [304].log_data[9].valid := 1, [304].log_data[10].valid := 1, [304].log_data[11].valid := 1, [304].log_data[12].valid := 1, [304].log_data[13].valid := 1, [304].log_data[14].valid := 1, [304].log_data[15].valid := 1, [304].log_data[16].valid := 1, [304].log_data[17].valid := 1, [304].log_data[18].valid := 1, [304].log_data[19].valid := 1, [304].time.Year := 2023, [304].time.Month := 1, [304].time.Day := 19, [304].time.Hour := 1, [304].time.Minute := 44, [304].time.Second := 59, [305].log_data[0].min := 1.0, [305].log_data[0].max := 1.0, [305].log_data[0].total := 300.0, [305].log_data[0].time := 300.0, [305].log_data[0].minminute := 45, [305].log_data[0].maxminute := 45, [305].log_data[0].valid := 1, [305].log_data[1].valid := 1, [305].log_data[2].valid := 1, [305].log_data[3].valid := 1, [305].log_data[4].valid := 1, [305].log_data[5].valid := 1, [305].log_data[6].valid := 1, [305].log_data[7].valid := 1, [305].log_data[8].valid := 1, [305].log_data[9].valid := 1, [305].log_data[10].valid := 1, [305].log_data[11].valid := 1, [305].log_data[12].valid := 1, [305].log_data[13].valid := 1, [305].log_data[14].valid := 1, [305].log_data[15].valid := 1, [305].log_data[16].valid := 1, [305].log_data[17].valid := 1, [305].log_data[18].valid := 1, [305].log_data[19].valid := 1, [305].time.Year := 2023, [305].time.Month := 1, [305].time.Day := 19, [305].time.Hour := 1,
        [305].time.Minute := 49, [305].time.Second := 59, [306].log_data[0].min := 1.0, [306].log_data[0].max := 1.0, [306].log_data[0].total := 300.0, [306].log_data[0].time := 300.0, [306].log_data[0].minminute := 50, [306].log_data[0].maxminute := 50, [306].log_data[0].valid := 1, [306].log_data[1].valid := 1, [306].log_data[2].valid := 1, [306].log_data[3].valid := 1, [306].log_data[4].valid := 1, [306].log_data[5].valid := 1, [306].log_data[6].valid := 1, [306].log_data[7].valid := 1, [306].log_data[8].valid := 1, [306].log_data[9].valid := 1, [306].log_data[10].valid := 1, [306].log_data[11].valid := 1, [306].log_data[12].valid := 1, [306].log_data[13].valid := 1, [306].log_data[14].valid := 1, [306].log_data[15].valid := 1, [306].log_data[16].valid := 1, [306].log_data[17].valid := 1, [306].log_data[18].valid := 1, [306].log_data[19].valid := 1, [306].time.Year := 2023, [306].time.Month := 1, [306].time.Day := 19, [306].time.Hour := 1, [306].time.Minute := 54, [306].time.Second := 59, [307].log_data[0].min := 1.0, [307].log_data[0].max := 1.0, [307].log_data[0].total := 300.0, [307].log_data[0].time := 300.0, [307].log_data[0].minminute := 55, [307].log_data[0].maxminute := 55, [307].log_data[0].valid := 1, [307].log_data[1].valid := 1, [307].log_data[2].valid := 1, [307].log_data[3].valid := 1, [307].log_data[4].valid := 1, [307].log_data[5].valid := 1, [307].log_data[6].valid := 1, [307].log_data[7].valid := 1, [307].log_data[8].valid := 1, [307].log_data[9].valid := 1, [307].log_data[10].valid := 1, [307].log_data[11].valid := 1, [307].log_data[12].valid := 1, [307].log_data[13].valid := 1, [307].log_data[14].valid := 1, [307].log_data[15].valid := 1, [307].log_data[16].valid := 1, [307].log_data[17].valid := 1, [307].log_data[18].valid := 1, [307].log_data[19].valid := 1,
        [307].time.Year := 2023, [307].time.Month := 1, [307].time.Day := 19, [307].time.Hour := 1, [307].time.Minute := 59, [307].time.Second := 59, [308].log_data[0].min := 1.0, [308].log_data[0].max := 1.0, [308].log_data[0].total := 300.0, [308].log_data[0].time := 300.0, [308].log_data[0].valid := 1, [308].log_data[1].valid := 1, [308].log_data[2].valid := 1, [308].log_data[3].valid := 1, [308].log_data[4].valid := 1, [308].log_data[5].valid := 1, [308].log_data[6].valid := 1, [308].log_data[7].valid := 1, [308].log_data[8].valid := 1, [308].log_data[9].valid := 1, [308].log_data[10].valid := 1, [308].log_data[11].valid := 1, [308].log_data[12].valid := 1, [308].log_data[13].valid := 1, [308].log_data[14].valid := 1, [308].log_data[15].valid := 1, [308].log_data[16].valid := 1, [308].log_data[17].valid := 1, [308].log_data[18].valid := 1, [308].log_data[19].valid := 1, [308].time.Year := 2023, [308].time.Month := 1, [308].time.Day := 19, [308].time.Hour := 2, [308].time.Minute := 4, [308].time.Second := 59, [309].log_data[0].min := 1.0, [309].log_data[0].max := 1.0, [309].log_data[0].total := 300.0, [309].log_data[0].time := 300.0, [309].log_data[0].minminute := 5, [309].log_data[0].maxminute := 5, [309].log_data[0].valid := 1, [309].log_data[1].valid := 1, [309].log_data[2].valid := 1, [309].log_data[3].valid := 1, [309].log_data[4].valid := 1, [309].log_data[5].valid := 1, [309].log_data[6].valid := 1, [309].log_data[7].valid := 1, [309].log_data[8].valid := 1, [309].log_data[9].valid := 1, [309].log_data[10].valid := 1, [309].log_data[11].valid := 1, [309].log_data[12].valid := 1, [309].log_data[13].valid := 1, [309].log_data[14].valid := 1, [309].log_data[15].valid := 1, [309].log_data[16].valid := 1, [309].log_data[17].valid := 1,
        [309].log_data[18].valid := 1, [309].log_data[19].valid := 1, [309].time.Year := 2023, [309].time.Month := 1, [309].time.Day := 19, [309].time.Hour := 2, [309].time.Minute := 9, [309].time.Second := 59, [310].log_data[0].min := 1.0, [310].log_data[0].max := 1.0, [310].log_data[0].total := 300.0, [310].log_data[0].time := 300.0, [310].log_data[0].minminute := 10, [310].log_data[0].maxminute := 10, [310].log_data[0].valid := 1, [310].log_data[1].valid := 1, [310].log_data[2].valid := 1, [310].log_data[3].valid := 1, [310].log_data[4].valid := 1, [310].log_data[5].valid := 1, [310].log_data[6].valid := 1, [310].log_data[7].valid := 1, [310].log_data[8].valid := 1, [310].log_data[9].valid := 1, [310].log_data[10].valid := 1, [310].log_data[11].valid := 1, [310].log_data[12].valid := 1, [310].log_data[13].valid := 1, [310].log_data[14].valid := 1, [310].log_data[15].valid := 1, [310].log_data[16].valid := 1, [310].log_data[17].valid := 1, [310].log_data[18].valid := 1, [310].log_data[19].valid := 1, [310].time.Year := 2023, [310].time.Month := 1, [310].time.Day := 19, [310].time.Hour := 2, [310].time.Minute := 14, [310].time.Second := 59, [311].log_data[0].min := 1.0, [311].log_data[0].max := 1.0, [311].log_data[0].total := 300.0, [311].log_data[0].time := 300.0, [311].log_data[0].minminute := 15, [311].log_data[0].maxminute := 15, [311].log_data[0].valid := 1, [311].log_data[1].valid := 1, [311].log_data[2].valid := 1, [311].log_data[3].valid := 1, [311].log_data[4].valid := 1, [311].log_data[5].valid := 1, [311].log_data[6].valid := 1, [311].log_data[7].valid := 1, [311].log_data[8].valid := 1, [311].log_data[9].valid := 1, [311].log_data[10].valid := 1, [311].log_data[11].valid := 1, [311].log_data[12].valid := 1, [311].log_data[13].valid := 1,
        [311].log_data[14].valid := 1, [311].log_data[15].valid := 1, [311].log_data[16].valid := 1, [311].log_data[17].valid := 1, [311].log_data[18].valid := 1, [311].log_data[19].valid := 1, [311].time.Year := 2023, [311].time.Month := 1, [311].time.Day := 19, [311].time.Hour := 2, [311].time.Minute := 19, [311].time.Second := 59, [312].log_data[0].min := 1.0, [312].log_data[0].max := 1.0, [312].log_data[0].total := 300.0, [312].log_data[0].time := 300.0, [312].log_data[0].minminute := 20, [312].log_data[0].maxminute := 20, [312].log_data[0].valid := 1, [312].log_data[1].valid := 1, [312].log_data[2].valid := 1, [312].log_data[3].valid := 1, [312].log_data[4].valid := 1, [312].log_data[5].valid := 1, [312].log_data[6].valid := 1, [312].log_data[7].valid := 1, [312].log_data[8].valid := 1, [312].log_data[9].valid := 1, [312].log_data[10].valid := 1, [312].log_data[11].valid := 1, [312].log_data[12].valid := 1, [312].log_data[13].valid := 1, [312].log_data[14].valid := 1, [312].log_data[15].valid := 1, [312].log_data[16].valid := 1, [312].log_data[17].valid := 1, [312].log_data[18].valid := 1, [312].log_data[19].valid := 1, [312].time.Year := 2023, [312].time.Month := 1, [312].time.Day := 19, [312].time.Hour := 2, [312].time.Minute := 24, [312].time.Second := 59, [313].log_data[0].min := 1.0, [313].log_data[0].max := 1.0, [313].log_data[0].total := 300.0, [313].log_data[0].time := 300.0, [313].log_data[0].minminute := 25, [313].log_data[0].maxminute := 25, [313].log_data[0].valid := 1, [313].log_data[1].valid := 1, [313].log_data[2].valid := 1, [313].log_data[3].valid := 1, [313].log_data[4].valid := 1, [313].log_data[5].valid := 1, [313].log_data[6].valid := 1, [313].log_data[7].valid := 1, [313].log_data[8].valid := 1, [313].log_data[9].valid := 1,
        [313].log_data[10].valid := 1, [313].log_data[11].valid := 1, [313].log_data[12].valid := 1, [313].log_data[13].valid := 1, [313].log_data[14].valid := 1, [313].log_data[15].valid := 1, [313].log_data[16].valid := 1, [313].log_data[17].valid := 1, [313].log_data[18].valid := 1, [313].log_data[19].valid := 1, [313].time.Year := 2023, [313].time.Month := 1, [313].time.Day := 19, [313].time.Hour := 2, [313].time.Minute := 29, [313].time.Second := 59, [314].log_data[0].min := 1.0, [314].log_data[0].max := 1.0, [314].log_data[0].total := 300.0, [314].log_data[0].time := 300.0, [314].log_data[0].minminute := 30, [314].log_data[0].maxminute := 30, [314].log_data[0].valid := 1, [314].log_data[1].valid := 1, [314].log_data[2].valid := 1, [314].log_data[3].valid := 1, [314].log_data[4].valid := 1, [314].log_data[5].valid := 1, [314].log_data[6].valid := 1, [314].log_data[7].valid := 1, [314].log_data[8].valid := 1, [314].log_data[9].valid := 1, [314].log_data[10].valid := 1, [314].log_data[11].valid := 1, [314].log_data[12].valid := 1, [314].log_data[13].valid := 1, [314].log_data[14].valid := 1, [314].log_data[15].valid := 1, [314].log_data[16].valid := 1, [314].log_data[17].valid := 1, [314].log_data[18].valid := 1, [314].log_data[19].valid := 1, [314].time.Year := 2023, [314].time.Month := 1, [314].time.Day := 19, [314].time.Hour := 2, [314].time.Minute := 34, [314].time.Second := 59, [315].log_data[0].min := 1.0, [315].log_data[0].max := 1.0, [315].log_data[0].total := 300.0, [315].log_data[0].time := 300.0, [315].log_data[0].minminute := 35, [315].log_data[0].maxminute := 35, [315].log_data[0].valid := 1, [315].log_data[1].valid := 1, [315].log_data[2].valid := 1, [315].log_data[3].valid := 1, [315].log_data[4].valid := 1, [315].log_data[5].valid := 1,
        [315].log_data[6].valid := 1, [315].log_data[7].valid := 1, [315].log_data[8].valid := 1, [315].log_data[9].valid := 1, [315].log_data[10].valid := 1, [315].log_data[11].valid := 1, [315].log_data[12].valid := 1, [315].log_data[13].valid := 1, [315].log_data[14].valid := 1, [315].log_data[15].valid := 1, [315].log_data[16].valid := 1, [315].log_data[17].valid := 1, [315].log_data[18].valid := 1, [315].log_data[19].valid := 1, [315].time.Year := 2023, [315].time.Month := 1, [315].time.Day := 19, [315].time.Hour := 2, [315].time.Minute := 39, [315].time.Second := 59, [316].log_data[0].min := 1.0, [316].log_data[0].max := 1.0, [316].log_data[0].total := 300.0, [316].log_data[0].time := 300.0, [316].log_data[0].minminute := 40, [316].log_data[0].maxminute := 40, [316].log_data[0].valid := 1, [316].log_data[1].valid := 1, [316].log_data[2].valid := 1, [316].log_data[3].valid := 1, [316].log_data[4].valid := 1, [316].log_data[5].valid := 1, [316].log_data[6].valid := 1, [316].log_data[7].valid := 1, [316].log_data[8].valid := 1, [316].log_data[9].valid := 1, [316].log_data[10].valid := 1, [316].log_data[11].valid := 1, [316].log_data[12].valid := 1, [316].log_data[13].valid := 1, [316].log_data[14].valid := 1, [316].log_data[15].valid := 1, [316].log_data[16].valid := 1, [316].log_data[17].valid := 1, [316].log_data[18].valid := 1, [316].log_data[19].valid := 1, [316].time.Year := 2023, [316].time.Month := 1, [316].time.Day := 19, [316].time.Hour := 2, [316].time.Minute := 44, [316].time.Second := 59, [317].log_data[0].min := 1.0, [317].log_data[0].max := 1.0, [317].log_data[0].total := 300.0, [317].log_data[0].time := 300.0, [317].log_data[0].minminute := 45, [317].log_data[0].maxminute := 45, [317].log_data[0].valid := 1, [317].log_data[1].valid := 1,
        [317].log_data[2].valid := 1, [317].log_data[3].valid := 1, [317].log_data[4].valid := 1, [317].log_data[5].valid := 1, [317].log_data[6].valid := 1, [317].log_data[7].valid := 1, [317].log_data[8].valid := 1, [317].log_data[9].valid := 1, [317].log_data[10].valid := 1, [317].log_data[11].valid := 1, [317].log_data[12].valid := 1, [317].log_data[13].valid := 1, [317].log_data[14].valid := 1, [317].log_data[15].valid := 1, [317].log_data[16].valid := 1, [317].log_data[17].valid := 1, [317].log_data[18].valid := 1, [317].log_data[19].valid := 1, [317].time.Year := 2023, [317].time.Month := 1, [317].time.Day := 19, [317].time.Hour := 2, [317].time.Minute := 49, [317].time.Second := 59, [318].log_data[0].min := 1.0, [318].log_data[0].max := 1.0, [318].log_data[0].total := 300.0, [318].log_data[0].time := 300.0, [318].log_data[0].minminute := 50, [318].log_data[0].maxminute := 50, [318].log_data[0].valid := 1, [318].log_data[1].valid := 1, [318].log_data[2].valid := 1, [318].log_data[3].valid := 1, [318].log_data[4].valid := 1, [318].log_data[5].valid := 1, [318].log_data[6].valid := 1, [318].log_data[7].valid := 1, [318].log_data[8].valid := 1, [318].log_data[9].valid := 1, [318].log_data[10].valid := 1, [318].log_data[11].valid := 1, [318].log_data[12].valid := 1, [318].log_data[13].valid := 1, [318].log_data[14].valid := 1, [318].log_data[15].valid := 1, [318].log_data[16].valid := 1, [318].log_data[17].valid := 1, [318].log_data[18].valid := 1, [318].log_data[19].valid := 1, [318].time.Year := 2023, [318].time.Month := 1, [318].time.Day := 19, [318].time.Hour := 2, [318].time.Minute := 54, [318].time.Second := 59, [319].log_data[0].min := 1.0, [319].log_data[0].max := 1.0, [319].log_data[0].total := 300.0, [319].log_data[0].time := 300.0,
        [319].log_data[0].minminute := 55, [319].log_data[0].maxminute := 55, [319].log_data[0].valid := 1, [319].log_data[1].valid := 1, [319].log_data[2].valid := 1, [319].log_data[3].valid := 1, [319].log_data[4].valid := 1, [319].log_data[5].valid := 1, [319].log_data[6].valid := 1, [319].log_data[7].valid := 1, [319].log_data[8].valid := 1, [319].log_data[9].valid := 1, [319].log_data[10].valid := 1, [319].log_data[11].valid := 1, [319].log_data[12].valid := 1, [319].log_data[13].valid := 1, [319].log_data[14].valid := 1, [319].log_data[15].valid := 1, [319].log_data[16].valid := 1, [319].log_data[17].valid := 1, [319].log_data[18].valid := 1, [319].log_data[19].valid := 1, [319].time.Year := 2023, [319].time.Month := 1, [319].time.Day := 19, [319].time.Hour := 2, [319].time.Minute := 59, [319].time.Second := 59, [320].log_data[0].min := 1.0, [320].log_data[0].max := 1.0, [320].log_data[0].total := 300.0, [320].log_data[0].time := 300.0, [320].log_data[0].valid := 1, [320].log_data[1].valid := 1, [320].log_data[2].valid := 1, [320].log_data[3].valid := 1, [320].log_data[4].valid := 1, [320].log_data[5].valid := 1, [320].log_data[6].valid := 1, [320].log_data[7].valid := 1, [320].log_data[8].valid := 1, [320].log_data[9].valid := 1, [320].log_data[10].valid := 1, [320].log_data[11].valid := 1, [320].log_data[12].valid := 1, [320].log_data[13].valid := 1, [320].log_data[14].valid := 1, [320].log_data[15].valid := 1, [320].log_data[16].valid := 1, [320].log_data[17].valid := 1, [320].log_data[18].valid := 1, [320].log_data[19].valid := 1, [320].time.Year := 2023, [320].time.Month := 1, [320].time.Day := 19, [320].time.Hour := 3, [320].time.Minute := 4, [320].time.Second := 59, [321].log_data[0].min := 1.0, [321].log_data[0].max := 1.0,
        [321].log_data[0].total := 300.0, [321].log_data[0].time := 300.0, [321].log_data[0].minminute := 5, [321].log_data[0].maxminute := 5, [321].log_data[0].valid := 1, [321].log_data[1].valid := 1, [321].log_data[2].valid := 1, [321].log_data[3].valid := 1, [321].log_data[4].valid := 1, [321].log_data[5].valid := 1, [321].log_data[6].valid := 1, [321].log_data[7].valid := 1, [321].log_data[8].valid := 1, [321].log_data[9].valid := 1, [321].log_data[10].valid := 1, [321].log_data[11].valid := 1, [321].log_data[12].valid := 1, [321].log_data[13].valid := 1, [321].log_data[14].valid := 1, [321].log_data[15].valid := 1, [321].log_data[16].valid := 1, [321].log_data[17].valid := 1, [321].log_data[18].valid := 1, [321].log_data[19].valid := 1, [321].time.Year := 2023, [321].time.Month := 1, [321].time.Day := 19, [321].time.Hour := 3, [321].time.Minute := 9, [321].time.Second := 59, [322].log_data[0].min := 1.0, [322].log_data[0].max := 1.0, [322].log_data[0].total := 300.0, [322].log_data[0].time := 300.0, [322].log_data[0].minminute := 10, [322].log_data[0].maxminute := 10, [322].log_data[0].valid := 1, [322].log_data[1].valid := 1, [322].log_data[2].valid := 1, [322].log_data[3].valid := 1, [322].log_data[4].valid := 1, [322].log_data[5].valid := 1, [322].log_data[6].valid := 1, [322].log_data[7].valid := 1, [322].log_data[8].valid := 1, [322].log_data[9].valid := 1, [322].log_data[10].valid := 1, [322].log_data[11].valid := 1, [322].log_data[12].valid := 1, [322].log_data[13].valid := 1, [322].log_data[14].valid := 1, [322].log_data[15].valid := 1, [322].log_data[16].valid := 1, [322].log_data[17].valid := 1, [322].log_data[18].valid := 1, [322].log_data[19].valid := 1, [322].time.Year := 2023, [322].time.Month := 1, [322].time.Day := 19, [322].time.Hour := 3,
        [322].time.Minute := 14, [322].time.Second := 59, [323].log_data[0].min := 1.0, [323].log_data[0].max := 1.0, [323].log_data[0].total := 300.0, [323].log_data[0].time := 300.0, [323].log_data[0].minminute := 15, [323].log_data[0].maxminute := 15, [323].log_data[0].valid := 1, [323].log_data[1].valid := 1, [323].log_data[2].valid := 1, [323].log_data[3].valid := 1, [323].log_data[4].valid := 1, [323].log_data[5].valid := 1, [323].log_data[6].valid := 1, [323].log_data[7].valid := 1, [323].log_data[8].valid := 1, [323].log_data[9].valid := 1, [323].log_data[10].valid := 1, [323].log_data[11].valid := 1, [323].log_data[12].valid := 1, [323].log_data[13].valid := 1, [323].log_data[14].valid := 1, [323].log_data[15].valid := 1, [323].log_data[16].valid := 1, [323].log_data[17].valid := 1, [323].log_data[18].valid := 1, [323].log_data[19].valid := 1, [323].time.Year := 2023, [323].time.Month := 1, [323].time.Day := 19, [323].time.Hour := 3, [323].time.Minute := 19, [323].time.Second := 59, [324].log_data[0].min := 1.0, [324].log_data[0].max := 1.0, [324].log_data[0].total := 300.0, [324].log_data[0].time := 300.0, [324].log_data[0].minminute := 20, [324].log_data[0].maxminute := 20, [324].log_data[0].valid := 1, [324].log_data[1].valid := 1, [324].log_data[2].valid := 1, [324].log_data[3].valid := 1, [324].log_data[4].valid := 1, [324].log_data[5].valid := 1, [324].log_data[6].valid := 1, [324].log_data[7].valid := 1, [324].log_data[8].valid := 1, [324].log_data[9].valid := 1, [324].log_data[10].valid := 1, [324].log_data[11].valid := 1, [324].log_data[12].valid := 1, [324].log_data[13].valid := 1, [324].log_data[14].valid := 1, [324].log_data[15].valid := 1, [324].log_data[16].valid := 1, [324].log_data[17].valid := 1, [324].log_data[18].valid := 1, [324].log_data[19].valid := 1,
        [324].time.Year := 2023, [324].time.Month := 1, [324].time.Day := 19, [324].time.Hour := 3, [324].time.Minute := 24, [324].time.Second := 59, [325].log_data[0].min := 1.0, [325].log_data[0].max := 1.0, [325].log_data[0].total := 300.0, [325].log_data[0].time := 300.0, [325].log_data[0].minminute := 25, [325].log_data[0].maxminute := 25, [325].log_data[0].valid := 1, [325].log_data[1].valid := 1, [325].log_data[2].valid := 1, [325].log_data[3].valid := 1, [325].log_data[4].valid := 1, [325].log_data[5].valid := 1, [325].log_data[6].valid := 1, [325].log_data[7].valid := 1, [325].log_data[8].valid := 1, [325].log_data[9].valid := 1, [325].log_data[10].valid := 1, [325].log_data[11].valid := 1, [325].log_data[12].valid := 1, [325].log_data[13].valid := 1, [325].log_data[14].valid := 1, [325].log_data[15].valid := 1, [325].log_data[16].valid := 1, [325].log_data[17].valid := 1, [325].log_data[18].valid := 1, [325].log_data[19].valid := 1, [325].time.Year := 2023, [325].time.Month := 1, [325].time.Day := 19, [325].time.Hour := 3, [325].time.Minute := 29, [325].time.Second := 59, [326].log_data[0].min := 1.0, [326].log_data[0].max := 1.0, [326].log_data[0].total := 300.0, [326].log_data[0].time := 300.0, [326].log_data[0].minminute := 30, [326].log_data[0].maxminute := 30, [326].log_data[0].valid := 1, [326].log_data[1].valid := 1, [326].log_data[2].valid := 1, [326].log_data[3].valid := 1, [326].log_data[4].valid := 1, [326].log_data[5].valid := 1, [326].log_data[6].valid := 1, [326].log_data[7].valid := 1, [326].log_data[8].valid := 1, [326].log_data[9].valid := 1, [326].log_data[10].valid := 1, [326].log_data[11].valid := 1, [326].log_data[12].valid := 1, [326].log_data[13].valid := 1, [326].log_data[14].valid := 1, [326].log_data[15].valid := 1,
        [326].log_data[16].valid := 1, [326].log_data[17].valid := 1, [326].log_data[18].valid := 1, [326].log_data[19].valid := 1, [326].time.Year := 2023, [326].time.Month := 1, [326].time.Day := 19, [326].time.Hour := 3, [326].time.Minute := 34, [326].time.Second := 59, [327].log_data[0].min := 1.0, [327].log_data[0].max := 1.0, [327].log_data[0].total := 300.0, [327].log_data[0].time := 300.0, [327].log_data[0].minminute := 35, [327].log_data[0].maxminute := 35, [327].log_data[0].valid := 1, [327].log_data[1].valid := 1, [327].log_data[2].valid := 1, [327].log_data[3].valid := 1, [327].log_data[4].valid := 1, [327].log_data[5].valid := 1, [327].log_data[6].valid := 1, [327].log_data[7].valid := 1, [327].log_data[8].valid := 1, [327].log_data[9].valid := 1, [327].log_data[10].valid := 1, [327].log_data[11].valid := 1, [327].log_data[12].valid := 1, [327].log_data[13].valid := 1, [327].log_data[14].valid := 1, [327].log_data[15].valid := 1, [327].log_data[16].valid := 1, [327].log_data[17].valid := 1, [327].log_data[18].valid := 1, [327].log_data[19].valid := 1, [327].time.Year := 2023, [327].time.Month := 1, [327].time.Day := 19, [327].time.Hour := 3, [327].time.Minute := 39, [327].time.Second := 59, [328].log_data[0].min := 1.0, [328].log_data[0].max := 1.0, [328].log_data[0].total := 300.0, [328].log_data[0].time := 300.0, [328].log_data[0].minminute := 40, [328].log_data[0].maxminute := 40, [328].log_data[0].valid := 1, [328].log_data[1].valid := 1, [328].log_data[2].valid := 1, [328].log_data[3].valid := 1, [328].log_data[4].valid := 1, [328].log_data[5].valid := 1, [328].log_data[6].valid := 1, [328].log_data[7].valid := 1, [328].log_data[8].valid := 1, [328].log_data[9].valid := 1, [328].log_data[10].valid := 1, [328].log_data[11].valid := 1,
        [328].log_data[12].valid := 1, [328].log_data[13].valid := 1, [328].log_data[14].valid := 1, [328].log_data[15].valid := 1, [328].log_data[16].valid := 1, [328].log_data[17].valid := 1, [328].log_data[18].valid := 1, [328].log_data[19].valid := 1, [328].time.Year := 2023, [328].time.Month := 1, [328].time.Day := 19, [328].time.Hour := 3, [328].time.Minute := 44, [328].time.Second := 59, [329].log_data[0].min := 1.0, [329].log_data[0].max := 1.0, [329].log_data[0].total := 300.0, [329].log_data[0].time := 300.0, [329].log_data[0].minminute := 45, [329].log_data[0].maxminute := 45, [329].log_data[0].valid := 1, [329].log_data[1].valid := 1, [329].log_data[2].valid := 1, [329].log_data[3].valid := 1, [329].log_data[4].valid := 1, [329].log_data[5].valid := 1, [329].log_data[6].valid := 1, [329].log_data[7].valid := 1, [329].log_data[8].valid := 1, [329].log_data[9].valid := 1, [329].log_data[10].valid := 1, [329].log_data[11].valid := 1, [329].log_data[12].valid := 1, [329].log_data[13].valid := 1, [329].log_data[14].valid := 1, [329].log_data[15].valid := 1, [329].log_data[16].valid := 1, [329].log_data[17].valid := 1, [329].log_data[18].valid := 1, [329].log_data[19].valid := 1, [329].time.Year := 2023, [329].time.Month := 1, [329].time.Day := 19, [329].time.Hour := 3, [329].time.Minute := 49, [329].time.Second := 59, [330].log_data[0].min := 1.0, [330].log_data[0].max := 1.0, [330].log_data[0].total := 300.0, [330].log_data[0].time := 300.0, [330].log_data[0].minminute := 50, [330].log_data[0].maxminute := 50, [330].log_data[0].valid := 1, [330].log_data[1].valid := 1, [330].log_data[2].valid := 1, [330].log_data[3].valid := 1, [330].log_data[4].valid := 1, [330].log_data[5].valid := 1, [330].log_data[6].valid := 1, [330].log_data[7].valid := 1,
        [330].log_data[8].valid := 1, [330].log_data[9].valid := 1, [330].log_data[10].valid := 1, [330].log_data[11].valid := 1, [330].log_data[12].valid := 1, [330].log_data[13].valid := 1, [330].log_data[14].valid := 1, [330].log_data[15].valid := 1, [330].log_data[16].valid := 1, [330].log_data[17].valid := 1, [330].log_data[18].valid := 1, [330].log_data[19].valid := 1, [330].time.Year := 2023, [330].time.Month := 1, [330].time.Day := 19, [330].time.Hour := 3, [330].time.Minute := 54, [330].time.Second := 59, [331].log_data[0].min := 1.0, [331].log_data[0].max := 1.0, [331].log_data[0].total := 300.0, [331].log_data[0].time := 300.0, [331].log_data[0].minminute := 55, [331].log_data[0].maxminute := 55, [331].log_data[0].valid := 1, [331].log_data[1].valid := 1, [331].log_data[2].valid := 1, [331].log_data[3].valid := 1, [331].log_data[4].valid := 1, [331].log_data[5].valid := 1, [331].log_data[6].valid := 1, [331].log_data[7].valid := 1, [331].log_data[8].valid := 1, [331].log_data[9].valid := 1, [331].log_data[10].valid := 1, [331].log_data[11].valid := 1, [331].log_data[12].valid := 1, [331].log_data[13].valid := 1, [331].log_data[14].valid := 1, [331].log_data[15].valid := 1, [331].log_data[16].valid := 1, [331].log_data[17].valid := 1, [331].log_data[18].valid := 1, [331].log_data[19].valid := 1, [331].time.Year := 2023, [331].time.Month := 1, [331].time.Day := 19, [331].time.Hour := 3, [331].time.Minute := 59, [331].time.Second := 59, [332].log_data[0].min := 1.0, [332].log_data[0].max := 1.0, [332].log_data[0].total := 300.0, [332].log_data[0].time := 300.0, [332].log_data[0].valid := 1, [332].log_data[1].valid := 1, [332].log_data[2].valid := 1, [332].log_data[3].valid := 1, [332].log_data[4].valid := 1, [332].log_data[5].valid := 1,
        [332].log_data[6].valid := 1, [332].log_data[7].valid := 1, [332].log_data[8].valid := 1, [332].log_data[9].valid := 1, [332].log_data[10].valid := 1, [332].log_data[11].valid := 1, [332].log_data[12].valid := 1, [332].log_data[13].valid := 1, [332].log_data[14].valid := 1, [332].log_data[15].valid := 1, [332].log_data[16].valid := 1, [332].log_data[17].valid := 1, [332].log_data[18].valid := 1, [332].log_data[19].valid := 1, [332].time.Year := 2023, [332].time.Month := 1, [332].time.Day := 19, [332].time.Hour := 4, [332].time.Minute := 4, [332].time.Second := 59, [333].log_data[0].min := 1.0, [333].log_data[0].max := 1.0, [333].log_data[0].total := 300.0, [333].log_data[0].time := 300.0, [333].log_data[0].minminute := 5, [333].log_data[0].maxminute := 5, [333].log_data[0].valid := 1, [333].log_data[1].valid := 1, [333].log_data[2].valid := 1, [333].log_data[3].valid := 1, [333].log_data[4].valid := 1, [333].log_data[5].valid := 1, [333].log_data[6].valid := 1, [333].log_data[7].valid := 1, [333].log_data[8].valid := 1, [333].log_data[9].valid := 1, [333].log_data[10].valid := 1, [333].log_data[11].valid := 1, [333].log_data[12].valid := 1, [333].log_data[13].valid := 1, [333].log_data[14].valid := 1, [333].log_data[15].valid := 1, [333].log_data[16].valid := 1, [333].log_data[17].valid := 1, [333].log_data[18].valid := 1, [333].log_data[19].valid := 1, [333].time.Year := 2023, [333].time.Month := 1, [333].time.Day := 19, [333].time.Hour := 4, [333].time.Minute := 9, [333].time.Second := 59, [334].log_data[0].min := 1.0, [334].log_data[0].max := 1.0, [334].log_data[0].total := 300.0, [334].log_data[0].time := 300.0, [334].log_data[0].minminute := 10, [334].log_data[0].maxminute := 10, [334].log_data[0].valid := 1, [334].log_data[1].valid := 1,
        [334].log_data[2].valid := 1, [334].log_data[3].valid := 1, [334].log_data[4].valid := 1, [334].log_data[5].valid := 1, [334].log_data[6].valid := 1, [334].log_data[7].valid := 1, [334].log_data[8].valid := 1, [334].log_data[9].valid := 1, [334].log_data[10].valid := 1, [334].log_data[11].valid := 1, [334].log_data[12].valid := 1, [334].log_data[13].valid := 1, [334].log_data[14].valid := 1, [334].log_data[15].valid := 1, [334].log_data[16].valid := 1, [334].log_data[17].valid := 1, [334].log_data[18].valid := 1, [334].log_data[19].valid := 1, [334].time.Year := 2023, [334].time.Month := 1, [334].time.Day := 19, [334].time.Hour := 4, [334].time.Minute := 14, [334].time.Second := 59, [335].log_data[0].min := 1.0, [335].log_data[0].max := 1.0, [335].log_data[0].total := 300.0, [335].log_data[0].time := 300.0, [335].log_data[0].minminute := 15, [335].log_data[0].maxminute := 15, [335].log_data[0].valid := 1, [335].log_data[1].valid := 1, [335].log_data[2].valid := 1, [335].log_data[3].valid := 1, [335].log_data[4].valid := 1, [335].log_data[5].valid := 1, [335].log_data[6].valid := 1, [335].log_data[7].valid := 1, [335].log_data[8].valid := 1, [335].log_data[9].valid := 1, [335].log_data[10].valid := 1, [335].log_data[11].valid := 1, [335].log_data[12].valid := 1, [335].log_data[13].valid := 1, [335].log_data[14].valid := 1, [335].log_data[15].valid := 1, [335].log_data[16].valid := 1, [335].log_data[17].valid := 1, [335].log_data[18].valid := 1, [335].log_data[19].valid := 1, [335].time.Year := 2023, [335].time.Month := 1, [335].time.Day := 19, [335].time.Hour := 4, [335].time.Minute := 19, [335].time.Second := 59, [336].log_data[0].min := 1.0, [336].log_data[0].max := 1.0, [336].log_data[0].total := 300.0, [336].log_data[0].time := 300.0,
        [336].log_data[0].minminute := 20, [336].log_data[0].maxminute := 20, [336].log_data[0].valid := 1, [336].log_data[1].valid := 1, [336].log_data[2].valid := 1, [336].log_data[3].valid := 1, [336].log_data[4].valid := 1, [336].log_data[5].valid := 1, [336].log_data[6].valid := 1, [336].log_data[7].valid := 1, [336].log_data[8].valid := 1, [336].log_data[9].valid := 1, [336].log_data[10].valid := 1, [336].log_data[11].valid := 1, [336].log_data[12].valid := 1, [336].log_data[13].valid := 1, [336].log_data[14].valid := 1, [336].log_data[15].valid := 1, [336].log_data[16].valid := 1, [336].log_data[17].valid := 1, [336].log_data[18].valid := 1, [336].log_data[19].valid := 1, [336].time.Year := 2023, [336].time.Month := 1, [336].time.Day := 19, [336].time.Hour := 4, [336].time.Minute := 24, [336].time.Second := 59, [337].log_data[0].min := 1.0, [337].log_data[0].max := 1.0, [337].log_data[0].total := 300.0, [337].log_data[0].time := 300.0, [337].log_data[0].minminute := 25, [337].log_data[0].maxminute := 25, [337].log_data[0].valid := 1, [337].log_data[1].valid := 1, [337].log_data[2].valid := 1, [337].log_data[3].valid := 1, [337].log_data[4].valid := 1, [337].log_data[5].valid := 1, [337].log_data[6].valid := 1, [337].log_data[7].valid := 1, [337].log_data[8].valid := 1, [337].log_data[9].valid := 1, [337].log_data[10].valid := 1, [337].log_data[11].valid := 1, [337].log_data[12].valid := 1, [337].log_data[13].valid := 1, [337].log_data[14].valid := 1, [337].log_data[15].valid := 1, [337].log_data[16].valid := 1, [337].log_data[17].valid := 1, [337].log_data[18].valid := 1, [337].log_data[19].valid := 1, [337].time.Year := 2023, [337].time.Month := 1, [337].time.Day := 19, [337].time.Hour := 4, [337].time.Minute := 29, [337].time.Second := 59,
        [338].log_data[0].min := 1.0, [338].log_data[0].max := 1.0, [338].log_data[0].total := 300.0, [338].log_data[0].time := 300.0, [338].log_data[0].minminute := 30, [338].log_data[0].maxminute := 30, [338].log_data[0].valid := 1, [338].log_data[1].valid := 1, [338].log_data[2].valid := 1, [338].log_data[3].valid := 1, [338].log_data[4].valid := 1, [338].log_data[5].valid := 1, [338].log_data[6].valid := 1, [338].log_data[7].valid := 1, [338].log_data[8].valid := 1, [338].log_data[9].valid := 1, [338].log_data[10].valid := 1, [338].log_data[11].valid := 1, [338].log_data[12].valid := 1, [338].log_data[13].valid := 1, [338].log_data[14].valid := 1, [338].log_data[15].valid := 1, [338].log_data[16].valid := 1, [338].log_data[17].valid := 1, [338].log_data[18].valid := 1, [338].log_data[19].valid := 1, [338].time.Year := 2023, [338].time.Month := 1, [338].time.Day := 19, [338].time.Hour := 4, [338].time.Minute := 34, [338].time.Second := 59, [339].log_data[0].min := 1.0, [339].log_data[0].max := 1.0, [339].log_data[0].total := 300.0, [339].log_data[0].time := 300.0, [339].log_data[0].minminute := 35, [339].log_data[0].maxminute := 35, [339].log_data[0].valid := 1, [339].log_data[1].valid := 1, [339].log_data[2].valid := 1, [339].log_data[3].valid := 1, [339].log_data[4].valid := 1, [339].log_data[5].valid := 1, [339].log_data[6].valid := 1, [339].log_data[7].valid := 1, [339].log_data[8].valid := 1, [339].log_data[9].valid := 1, [339].log_data[10].valid := 1, [339].log_data[11].valid := 1, [339].log_data[12].valid := 1, [339].log_data[13].valid := 1, [339].log_data[14].valid := 1, [339].log_data[15].valid := 1, [339].log_data[16].valid := 1, [339].log_data[17].valid := 1, [339].log_data[18].valid := 1, [339].log_data[19].valid := 1, [339].time.Year := 2023, [339].time.Month := 1,
        [339].time.Day := 19, [339].time.Hour := 4, [339].time.Minute := 39, [339].time.Second := 59, [340].log_data[0].min := 1.0, [340].log_data[0].max := 1.0, [340].log_data[0].total := 300.0, [340].log_data[0].time := 300.0, [340].log_data[0].minminute := 40, [340].log_data[0].maxminute := 40, [340].log_data[0].valid := 1, [340].log_data[1].valid := 1, [340].log_data[2].valid := 1, [340].log_data[3].valid := 1, [340].log_data[4].valid := 1, [340].log_data[5].valid := 1, [340].log_data[6].valid := 1, [340].log_data[7].valid := 1, [340].log_data[8].valid := 1, [340].log_data[9].valid := 1, [340].log_data[10].valid := 1, [340].log_data[11].valid := 1, [340].log_data[12].valid := 1, [340].log_data[13].valid := 1, [340].log_data[14].valid := 1, [340].log_data[15].valid := 1, [340].log_data[16].valid := 1, [340].log_data[17].valid := 1, [340].log_data[18].valid := 1, [340].log_data[19].valid := 1, [340].time.Year := 2023, [340].time.Month := 1, [340].time.Day := 19, [340].time.Hour := 4, [340].time.Minute := 44, [340].time.Second := 59, [341].log_data[0].min := 1.0, [341].log_data[0].max := 1.0, [341].log_data[0].total := 300.0, [341].log_data[0].time := 300.0, [341].log_data[0].minminute := 45, [341].log_data[0].maxminute := 45, [341].log_data[0].valid := 1, [341].log_data[1].valid := 1, [341].log_data[2].valid := 1, [341].log_data[3].valid := 1, [341].log_data[4].valid := 1, [341].log_data[5].valid := 1, [341].log_data[6].valid := 1, [341].log_data[7].valid := 1, [341].log_data[8].valid := 1, [341].log_data[9].valid := 1, [341].log_data[10].valid := 1, [341].log_data[11].valid := 1, [341].log_data[12].valid := 1, [341].log_data[13].valid := 1, [341].log_data[14].valid := 1, [341].log_data[15].valid := 1, [341].log_data[16].valid := 1, [341].log_data[17].valid := 1,
        [341].log_data[18].valid := 1, [341].log_data[19].valid := 1, [341].time.Year := 2023, [341].time.Month := 1, [341].time.Day := 19, [341].time.Hour := 4, [341].time.Minute := 49, [341].time.Second := 59, [342].log_data[0].min := 1.0, [342].log_data[0].max := 1.0, [342].log_data[0].total := 300.0, [342].log_data[0].time := 300.0, [342].log_data[0].minminute := 50, [342].log_data[0].maxminute := 50, [342].log_data[0].valid := 1, [342].log_data[1].valid := 1, [342].log_data[2].valid := 1, [342].log_data[3].valid := 1, [342].log_data[4].valid := 1, [342].log_data[5].valid := 1, [342].log_data[6].valid := 1, [342].log_data[7].valid := 1, [342].log_data[8].valid := 1, [342].log_data[9].valid := 1, [342].log_data[10].valid := 1, [342].log_data[11].valid := 1, [342].log_data[12].valid := 1, [342].log_data[13].valid := 1, [342].log_data[14].valid := 1, [342].log_data[15].valid := 1, [342].log_data[16].valid := 1, [342].log_data[17].valid := 1, [342].log_data[18].valid := 1, [342].log_data[19].valid := 1, [342].time.Year := 2023, [342].time.Month := 1, [342].time.Day := 19, [342].time.Hour := 4, [342].time.Minute := 54, [342].time.Second := 59, [343].log_data[0].min := 1.0, [343].log_data[0].max := 1.0, [343].log_data[0].total := 300.0, [343].log_data[0].time := 300.0, [343].log_data[0].minminute := 55, [343].log_data[0].maxminute := 55, [343].log_data[0].valid := 1, [343].log_data[1].valid := 1, [343].log_data[2].valid := 1, [343].log_data[3].valid := 1, [343].log_data[4].valid := 1, [343].log_data[5].valid := 1, [343].log_data[6].valid := 1, [343].log_data[7].valid := 1, [343].log_data[8].valid := 1, [343].log_data[9].valid := 1, [343].log_data[10].valid := 1, [343].log_data[11].valid := 1, [343].log_data[12].valid := 1, [343].log_data[13].valid := 1,
        [343].log_data[14].valid := 1, [343].log_data[15].valid := 1, [343].log_data[16].valid := 1, [343].log_data[17].valid := 1, [343].log_data[18].valid := 1, [343].log_data[19].valid := 1, [343].time.Year := 2023, [343].time.Month := 1, [343].time.Day := 19, [343].time.Hour := 4, [343].time.Minute := 59, [343].time.Second := 59, [344].log_data[0].min := 1.0, [344].log_data[0].max := 1.0, [344].log_data[0].total := 300.0, [344].log_data[0].time := 300.0, [344].log_data[0].valid := 1, [344].log_data[1].valid := 1, [344].log_data[2].valid := 1, [344].log_data[3].valid := 1, [344].log_data[4].valid := 1, [344].log_data[5].valid := 1, [344].log_data[6].valid := 1, [344].log_data[7].valid := 1, [344].log_data[8].valid := 1, [344].log_data[9].valid := 1, [344].log_data[10].valid := 1, [344].log_data[11].valid := 1, [344].log_data[12].valid := 1, [344].log_data[13].valid := 1, [344].log_data[14].valid := 1, [344].log_data[15].valid := 1, [344].log_data[16].valid := 1, [344].log_data[17].valid := 1, [344].log_data[18].valid := 1, [344].log_data[19].valid := 1, [344].time.Year := 2023, [344].time.Month := 1, [344].time.Day := 19, [344].time.Hour := 5, [344].time.Minute := 4, [344].time.Second := 59, [345].log_data[0].min := 1.0, [345].log_data[0].max := 1.0, [345].log_data[0].total := 300.0, [345].log_data[0].time := 300.0, [345].log_data[0].minminute := 5, [345].log_data[0].maxminute := 5, [345].log_data[0].valid := 1, [345].log_data[1].valid := 1, [345].log_data[2].valid := 1, [345].log_data[3].valid := 1, [345].log_data[4].valid := 1, [345].log_data[5].valid := 1, [345].log_data[6].valid := 1, [345].log_data[7].valid := 1, [345].log_data[8].valid := 1, [345].log_data[9].valid := 1, [345].log_data[10].valid := 1, [345].log_data[11].valid := 1,
        [345].log_data[12].valid := 1, [345].log_data[13].valid := 1, [345].log_data[14].valid := 1, [345].log_data[15].valid := 1, [345].log_data[16].valid := 1, [345].log_data[17].valid := 1, [345].log_data[18].valid := 1, [345].log_data[19].valid := 1, [345].time.Year := 2023, [345].time.Month := 1, [345].time.Day := 19, [345].time.Hour := 5, [345].time.Minute := 9, [345].time.Second := 59, [346].log_data[0].min := 1.0, [346].log_data[0].max := 1.0, [346].log_data[0].total := 300.0, [346].log_data[0].time := 300.0, [346].log_data[0].minminute := 10, [346].log_data[0].maxminute := 10, [346].log_data[0].valid := 1, [346].log_data[1].valid := 1, [346].log_data[2].valid := 1, [346].log_data[3].valid := 1, [346].log_data[4].valid := 1, [346].log_data[5].valid := 1, [346].log_data[6].valid := 1, [346].log_data[7].valid := 1, [346].log_data[8].valid := 1, [346].log_data[9].valid := 1, [346].log_data[10].valid := 1, [346].log_data[11].valid := 1, [346].log_data[12].valid := 1, [346].log_data[13].valid := 1, [346].log_data[14].valid := 1, [346].log_data[15].valid := 1, [346].log_data[16].valid := 1, [346].log_data[17].valid := 1, [346].log_data[18].valid := 1, [346].log_data[19].valid := 1, [346].time.Year := 2023, [346].time.Month := 1, [346].time.Day := 19, [346].time.Hour := 5, [346].time.Minute := 14, [346].time.Second := 59, [347].log_data[0].min := 1.0, [347].log_data[0].max := 1.0, [347].log_data[0].total := 300.0, [347].log_data[0].time := 300.0, [347].log_data[0].minminute := 15, [347].log_data[0].maxminute := 15, [347].log_data[0].valid := 1, [347].log_data[1].valid := 1, [347].log_data[2].valid := 1, [347].log_data[3].valid := 1, [347].log_data[4].valid := 1, [347].log_data[5].valid := 1, [347].log_data[6].valid := 1, [347].log_data[7].valid := 1,
        [347].log_data[8].valid := 1, [347].log_data[9].valid := 1, [347].log_data[10].valid := 1, [347].log_data[11].valid := 1, [347].log_data[12].valid := 1, [347].log_data[13].valid := 1, [347].log_data[14].valid := 1, [347].log_data[15].valid := 1, [347].log_data[16].valid := 1, [347].log_data[17].valid := 1, [347].log_data[18].valid := 1, [347].log_data[19].valid := 1, [347].time.Year := 2023, [347].time.Month := 1, [347].time.Day := 19, [347].time.Hour := 5, [347].time.Minute := 19, [347].time.Second := 59, [348].log_data[0].min := 1.0, [348].log_data[0].max := 1.0, [348].log_data[0].total := 300.0, [348].log_data[0].time := 300.0, [348].log_data[0].minminute := 20, [348].log_data[0].maxminute := 20, [348].log_data[0].valid := 1, [348].log_data[1].valid := 1, [348].log_data[2].valid := 1, [348].log_data[3].valid := 1, [348].log_data[4].valid := 1, [348].log_data[5].valid := 1, [348].log_data[6].valid := 1, [348].log_data[7].valid := 1, [348].log_data[8].valid := 1, [348].log_data[9].valid := 1, [348].log_data[10].valid := 1, [348].log_data[11].valid := 1, [348].log_data[12].valid := 1, [348].log_data[13].valid := 1, [348].log_data[14].valid := 1, [348].log_data[15].valid := 1, [348].log_data[16].valid := 1, [348].log_data[17].valid := 1, [348].log_data[18].valid := 1, [348].log_data[19].valid := 1, [348].time.Year := 2023, [348].time.Month := 1, [348].time.Day := 19, [348].time.Hour := 5, [348].time.Minute := 24, [348].time.Second := 59, [349].log_data[0].min := 1.0, [349].log_data[0].max := 1.0, [349].log_data[0].total := 300.0, [349].log_data[0].time := 300.0, [349].log_data[0].minminute := 25, [349].log_data[0].maxminute := 25, [349].log_data[0].valid := 1, [349].log_data[1].valid := 1, [349].log_data[2].valid := 1, [349].log_data[3].valid := 1,
        [349].log_data[4].valid := 1, [349].log_data[5].valid := 1, [349].log_data[6].valid := 1, [349].log_data[7].valid := 1, [349].log_data[8].valid := 1, [349].log_data[9].valid := 1, [349].log_data[10].valid := 1, [349].log_data[11].valid := 1, [349].log_data[12].valid := 1, [349].log_data[13].valid := 1, [349].log_data[14].valid := 1, [349].log_data[15].valid := 1, [349].log_data[16].valid := 1, [349].log_data[17].valid := 1, [349].log_data[18].valid := 1, [349].log_data[19].valid := 1, [349].time.Year := 2023, [349].time.Month := 1, [349].time.Day := 19, [349].time.Hour := 5, [349].time.Minute := 29, [349].time.Second := 59, [350].log_data[0].min := 1.0, [350].log_data[0].max := 1.0, [350].log_data[0].total := 300.0, [350].log_data[0].time := 300.0, [350].log_data[0].minminute := 30, [350].log_data[0].maxminute := 30, [350].log_data[0].valid := 1, [350].log_data[1].valid := 1, [350].log_data[2].valid := 1, [350].log_data[3].valid := 1, [350].log_data[4].valid := 1, [350].log_data[5].valid := 1, [350].log_data[6].valid := 1, [350].log_data[7].valid := 1, [350].log_data[8].valid := 1, [350].log_data[9].valid := 1, [350].log_data[10].valid := 1, [350].log_data[11].valid := 1, [350].log_data[12].valid := 1, [350].log_data[13].valid := 1, [350].log_data[14].valid := 1, [350].log_data[15].valid := 1, [350].log_data[16].valid := 1, [350].log_data[17].valid := 1, [350].log_data[18].valid := 1, [350].log_data[19].valid := 1, [350].time.Year := 2023, [350].time.Month := 1, [350].time.Day := 19, [350].time.Hour := 5, [350].time.Minute := 34, [350].time.Second := 59, [351].log_data[0].min := 1.0, [351].log_data[0].max := 1.0, [351].log_data[0].total := 300.0, [351].log_data[0].time := 300.0, [351].log_data[0].minminute := 35, [351].log_data[0].maxminute := 35,
        [351].log_data[0].valid := 1, [351].log_data[1].valid := 1, [351].log_data[2].valid := 1, [351].log_data[3].valid := 1, [351].log_data[4].valid := 1, [351].log_data[5].valid := 1, [351].log_data[6].valid := 1, [351].log_data[7].valid := 1, [351].log_data[8].valid := 1, [351].log_data[9].valid := 1, [351].log_data[10].valid := 1, [351].log_data[11].valid := 1, [351].log_data[12].valid := 1, [351].log_data[13].valid := 1, [351].log_data[14].valid := 1, [351].log_data[15].valid := 1, [351].log_data[16].valid := 1, [351].log_data[17].valid := 1, [351].log_data[18].valid := 1, [351].log_data[19].valid := 1, [351].time.Year := 2023, [351].time.Month := 1, [351].time.Day := 19, [351].time.Hour := 5, [351].time.Minute := 39, [351].time.Second := 59, [352].log_data[0].min := 1.0, [352].log_data[0].max := 1.0, [352].log_data[0].total := 300.0, [352].log_data[0].time := 300.0, [352].log_data[0].minminute := 40, [352].log_data[0].maxminute := 40, [352].log_data[0].valid := 1, [352].log_data[1].valid := 1, [352].log_data[2].valid := 1, [352].log_data[3].valid := 1, [352].log_data[4].valid := 1, [352].log_data[5].valid := 1, [352].log_data[6].valid := 1, [352].log_data[7].valid := 1, [352].log_data[8].valid := 1, [352].log_data[9].valid := 1, [352].log_data[10].valid := 1, [352].log_data[11].valid := 1, [352].log_data[12].valid := 1, [352].log_data[13].valid := 1, [352].log_data[14].valid := 1, [352].log_data[15].valid := 1, [352].log_data[16].valid := 1, [352].log_data[17].valid := 1, [352].log_data[18].valid := 1, [352].log_data[19].valid := 1, [352].time.Year := 2023, [352].time.Month := 1, [352].time.Day := 19, [352].time.Hour := 5, [352].time.Minute := 44, [352].time.Second := 59, [353].log_data[0].min := 1.0, [353].log_data[0].max := 1.0,
        [353].log_data[0].total := 300.0, [353].log_data[0].time := 300.0, [353].log_data[0].minminute := 45, [353].log_data[0].maxminute := 45, [353].log_data[0].valid := 1, [353].log_data[1].valid := 1, [353].log_data[2].valid := 1, [353].log_data[3].valid := 1, [353].log_data[4].valid := 1, [353].log_data[5].valid := 1, [353].log_data[6].valid := 1, [353].log_data[7].valid := 1, [353].log_data[8].valid := 1, [353].log_data[9].valid := 1, [353].log_data[10].valid := 1, [353].log_data[11].valid := 1, [353].log_data[12].valid := 1, [353].log_data[13].valid := 1, [353].log_data[14].valid := 1, [353].log_data[15].valid := 1, [353].log_data[16].valid := 1, [353].log_data[17].valid := 1, [353].log_data[18].valid := 1, [353].log_data[19].valid := 1, [353].time.Year := 2023, [353].time.Month := 1, [353].time.Day := 19, [353].time.Hour := 5, [353].time.Minute := 49, [353].time.Second := 59, [354].log_data[0].min := 1.0, [354].log_data[0].max := 1.0, [354].log_data[0].total := 300.0, [354].log_data[0].time := 300.0, [354].log_data[0].minminute := 50, [354].log_data[0].maxminute := 50, [354].log_data[0].valid := 1, [354].log_data[1].valid := 1, [354].log_data[2].valid := 1, [354].log_data[3].valid := 1, [354].log_data[4].valid := 1, [354].log_data[5].valid := 1, [354].log_data[6].valid := 1, [354].log_data[7].valid := 1, [354].log_data[8].valid := 1, [354].log_data[9].valid := 1, [354].log_data[10].valid := 1, [354].log_data[11].valid := 1, [354].log_data[12].valid := 1, [354].log_data[13].valid := 1, [354].log_data[14].valid := 1, [354].log_data[15].valid := 1, [354].log_data[16].valid := 1, [354].log_data[17].valid := 1, [354].log_data[18].valid := 1, [354].log_data[19].valid := 1, [354].time.Year := 2023, [354].time.Month := 1, [354].time.Day := 19, [354].time.Hour := 5,
        [354].time.Minute := 54, [354].time.Second := 59, [355].log_data[0].min := 1.0, [355].log_data[0].max := 1.0, [355].log_data[0].total := 300.0, [355].log_data[0].time := 300.0, [355].log_data[0].minminute := 55, [355].log_data[0].maxminute := 55, [355].log_data[0].valid := 1, [355].log_data[1].valid := 1, [355].log_data[2].valid := 1, [355].log_data[3].valid := 1, [355].log_data[4].valid := 1, [355].log_data[5].valid := 1, [355].log_data[6].valid := 1, [355].log_data[7].valid := 1, [355].log_data[8].valid := 1, [355].log_data[9].valid := 1, [355].log_data[10].valid := 1, [355].log_data[11].valid := 1, [355].log_data[12].valid := 1, [355].log_data[13].valid := 1, [355].log_data[14].valid := 1, [355].log_data[15].valid := 1, [355].log_data[16].valid := 1, [355].log_data[17].valid := 1, [355].log_data[18].valid := 1, [355].log_data[19].valid := 1, [355].time.Year := 2023, [355].time.Month := 1, [355].time.Day := 19, [355].time.Hour := 5, [355].time.Minute := 59, [355].time.Second := 59, [356].log_data[0].min := 1.0, [356].log_data[0].max := 1.0, [356].log_data[0].total := 300.0, [356].log_data[0].time := 300.0, [356].log_data[0].valid := 1, [356].log_data[1].valid := 1, [356].log_data[2].valid := 1, [356].log_data[3].valid := 1, [356].log_data[4].valid := 1, [356].log_data[5].valid := 1, [356].log_data[6].valid := 1, [356].log_data[7].valid := 1, [356].log_data[8].valid := 1, [356].log_data[9].valid := 1, [356].log_data[10].valid := 1, [356].log_data[11].valid := 1, [356].log_data[12].valid := 1, [356].log_data[13].valid := 1, [356].log_data[14].valid := 1, [356].log_data[15].valid := 1, [356].log_data[16].valid := 1, [356].log_data[17].valid := 1, [356].log_data[18].valid := 1, [356].log_data[19].valid := 1, [356].time.Year := 2023, [356].time.Month := 1,
        [356].time.Day := 19, [356].time.Hour := 6, [356].time.Minute := 4, [356].time.Second := 59, [357].log_data[0].min := 1.0, [357].log_data[0].max := 1.0, [357].log_data[0].total := 300.0, [357].log_data[0].time := 300.0, [357].log_data[0].minminute := 5, [357].log_data[0].maxminute := 5, [357].log_data[0].valid := 1, [357].log_data[1].valid := 1, [357].log_data[2].valid := 1, [357].log_data[3].valid := 1, [357].log_data[4].valid := 1, [357].log_data[5].valid := 1, [357].log_data[6].valid := 1, [357].log_data[7].valid := 1, [357].log_data[8].valid := 1, [357].log_data[9].valid := 1, [357].log_data[10].valid := 1, [357].log_data[11].valid := 1, [357].log_data[12].valid := 1, [357].log_data[13].valid := 1, [357].log_data[14].valid := 1, [357].log_data[15].valid := 1, [357].log_data[16].valid := 1, [357].log_data[17].valid := 1, [357].log_data[18].valid := 1, [357].log_data[19].valid := 1, [357].time.Year := 2023, [357].time.Month := 1, [357].time.Day := 19, [357].time.Hour := 6, [357].time.Minute := 9, [357].time.Second := 59, [358].log_data[0].min := 1.0, [358].log_data[0].max := 1.0, [358].log_data[0].total := 300.0, [358].log_data[0].time := 300.0, [358].log_data[0].minminute := 10, [358].log_data[0].maxminute := 10, [358].log_data[0].valid := 1, [358].log_data[1].valid := 1, [358].log_data[2].valid := 1, [358].log_data[3].valid := 1, [358].log_data[4].valid := 1, [358].log_data[5].valid := 1, [358].log_data[6].valid := 1, [358].log_data[7].valid := 1, [358].log_data[8].valid := 1, [358].log_data[9].valid := 1, [358].log_data[10].valid := 1, [358].log_data[11].valid := 1, [358].log_data[12].valid := 1, [358].log_data[13].valid := 1, [358].log_data[14].valid := 1, [358].log_data[15].valid := 1, [358].log_data[16].valid := 1, [358].log_data[17].valid := 1,
        [358].log_data[18].valid := 1, [358].log_data[19].valid := 1, [358].time.Year := 2023, [358].time.Month := 1, [358].time.Day := 19, [358].time.Hour := 6, [358].time.Minute := 14, [358].time.Second := 59, [359].log_data[0].min := 1.0, [359].log_data[0].max := 1.0, [359].log_data[0].total := 300.0, [359].log_data[0].time := 300.0, [359].log_data[0].minminute := 15, [359].log_data[0].maxminute := 15, [359].log_data[0].valid := 1, [359].log_data[1].valid := 1, [359].log_data[2].valid := 1, [359].log_data[3].valid := 1, [359].log_data[4].valid := 1, [359].log_data[5].valid := 1, [359].log_data[6].valid := 1, [359].log_data[7].valid := 1, [359].log_data[8].valid := 1, [359].log_data[9].valid := 1, [359].log_data[10].valid := 1, [359].log_data[11].valid := 1, [359].log_data[12].valid := 1, [359].log_data[13].valid := 1, [359].log_data[14].valid := 1, [359].log_data[15].valid := 1, [359].log_data[16].valid := 1, [359].log_data[17].valid := 1, [359].log_data[18].valid := 1, [359].log_data[19].valid := 1, [359].time.Year := 2023, [359].time.Month := 1, [359].time.Day := 19, [359].time.Hour := 6, [359].time.Minute := 19, [359].time.Second := 59, [360].log_data[0].min := 1.0, [360].log_data[0].max := 1.0, [360].log_data[0].total := 300.0, [360].log_data[0].time := 300.0, [360].log_data[0].minminute := 20, [360].log_data[0].maxminute := 20, [360].log_data[0].valid := 1, [360].log_data[1].valid := 1, [360].log_data[2].valid := 1, [360].log_data[3].valid := 1, [360].log_data[4].valid := 1, [360].log_data[5].valid := 1, [360].log_data[6].valid := 1, [360].log_data[7].valid := 1, [360].log_data[8].valid := 1, [360].log_data[9].valid := 1, [360].log_data[10].valid := 1, [360].log_data[11].valid := 1, [360].log_data[12].valid := 1, [360].log_data[13].valid := 1,
